KUKA KRL program: EPS_2_251806_MH03A_A_20260213065131.src

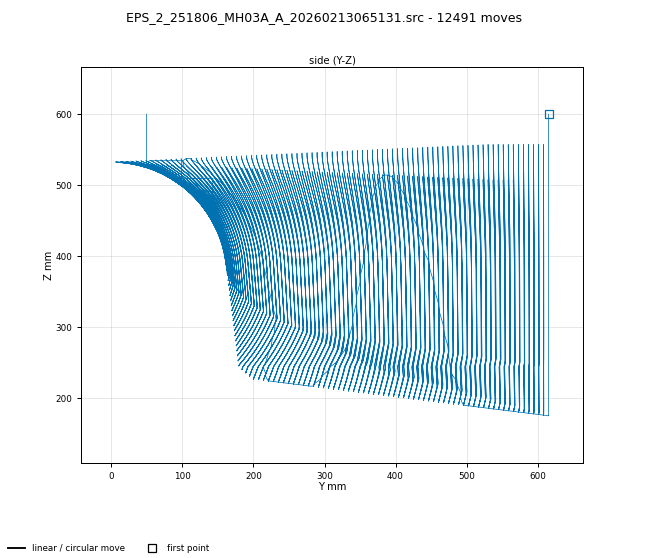
[picture p0: tool path of EPS_2_251806_MH03A_A_20260213065131.src, 12491 of 12493 moves have a stored position in this frame; points joined in program order, loops and branches not executed]
&ACCESS RVP
&REL 4
&COMMENT QRS 19112012
&PARAM EDITMASK = *
DEF PART()
EXT BAS (BAS_COMMAND :IN,REAL :IN )
INT I
BAS (#INITMOV,0 )

;KUKA QRS Post kuka4.cps  Date:22-06-2017 !

File_ID=3027

QRS_PRE_INIT()

;Init var - Until changes are made in qrs_pre_init
Outlet_Square_prg=0
Inlet_1_Square_prg=0
Inlet_2_Square_prg=0
Inlet_3_Square_prg=0
Inlet_4_Square_prg=0
Inlet_5_Square_prg=0

Outlet_1={X 0.000, Y 529.100, Z 408.000, B 0.000, E1 0.000 }
Inlet_1={X 0.000, Y 536.530, Z 382.000, B 0.000, E1 180.000 }
Outlet_1_type=299
Inlet_1_type=251
;QRS#1=Sidecore dimensions
;QRS#2=300-12" PVC SDR 35
;QRS#3=250-10" PVC SDR 35
;QRS#4=
;QRS#5=
;QRS#6=
;QRS#7=
;QRS#8=
;QRS#9=16M PSX
;QRS#10=14M PSX
;QRS#11=
;QRS#12=
;QRS#13=
;QRS#14=
;QRS#15=
;QRS#16=1220x127x838 2,75'
;QRS#17=EPS Height
;QRS#18=557,5
;QRS#19=*
;QRS#20= UPDATED VERSION 22-06-2017
;QRS#21=*
Outlet_Square=0150
Inlet_1_Square=0100
Inlet_2_Square=0
Inlet_3_Square=0
Inlet_4_Square=0
Inlet_5_Square=0
Mill_Square=1
Outlet_Square_Prg=206
Inlet_1_Square_prg=205

QRS_INIT()

$ADVANCE=5

; T1
PTP {E1 173.606,E2 173.606}
PTP {X 0,Y 615.5,A -85,B 0,C 180,E1 173.606,E2 173.606,E3 0,E4 0,E5 0,E6 0}
QRS_SPEED_INIT()
LIN {X 0,Y 615.5,Z 600,A -85,B 0,C 180,E1 173.606,E2 173.606,E3 0,E4 0,E5 0,E6 0} C_VEL
LIN {X 0,Y 615.5,Z 185.489,A -85,B 0,C 180,E1 173.606,E2 173.606} C_VEL
LIN {X 0,Y 615.5,Z 177.309,A -85,B 0,C 180,E1 173.606,E2 173.606} C_VEL
LIN {X 0,Y 615.485,Z 175.309,A -85,B 0,C 180,E1 173.419,E2 173.419} C_VEL
LIN {X 0,Y 615.484,Z 175.321,A -85,B 0,C 180,E1 170.801,E2 170.801} C_VEL
LIN {X 0,Y 615.479,Z 175.314,A -85,B 0,C 180,E1 168.139,E2 168.139} C_VEL
LIN {X 0,Y 615.481,Z 175.311,A -85,B 0,C 180,E1 165.451,E2 165.451} C_VEL
LIN {X 0,Y 615.493,Z 175.325,A -85,B 0,C 180,E1 162.73,E2 162.73} C_VEL
LIN {X 0,Y 615.49,Z 175.308,A -85,B 0,C 180,E1 159.967,E2 159.967} C_VEL
LIN {X 0,Y 615.483,Z 175.321,A -85,B 0,C 180,E1 157.155,E2 157.155} C_VEL
LIN {X 0,Y 615.475,Z 175.315,A -85,B 0,C 180,E1 154.433,E2 154.433} C_VEL
LIN {X 0,Y 615.483,Z 175.309,A -85,B 0,C 180,E1 152.085,E2 152.085} C_VEL
LIN {X 0,Y 615.492,Z 175.326,A -85,B 0,C 180,E1 149.08,E2 149.08} C_VEL
LIN {X 0,Y 615.474,Z 175.312,A -85,B 0,C 180,E1 146.467,E2 146.467} C_VEL
LIN {X 0,Y 615.492,Z 175.307,A -85,B 0,C 180,E1 144.165,E2 144.165} C_VEL
LIN {X 0,Y 615.485,Z 175.311,A -85,B 0,C 180,E1 141.931,E2 141.931} C_VEL
LIN {X 0,Y 615.486,Z 175.327,A -85,B 0,C 180,E1 139.393,E2 139.393} C_VEL
LIN {X 0,Y 615.469,Z 175.314,A -85,B 0,C 180,E1 136.753,E2 136.753} C_VEL
LIN {X 0,Y 615.488,Z 175.312,A -85,B 0,C 180,E1 133.997,E2 133.997} C_VEL
LIN {X 0,Y 615.49,Z 175.325,A -85,B 0,C 180,E1 131.473,E2 131.473} C_VEL
LIN {X 0,Y 615.465,Z 175.315,A -85,B 0,C 180,E1 128.906,E2 128.906} C_VEL
LIN {X 0,Y 615.484,Z 175.31,A -85,B 0,C 180,E1 126.425,E2 126.425} C_VEL
LIN {X 0,Y 615.481,Z 175.322,A -85,B 0,C 180,E1 123.533,E2 123.533} C_VEL
LIN {X 0,Y 615.466,Z 175.313,A -85,B 0,C 180,E1 120.921,E2 120.921} C_VEL
LIN {X 0,Y 615.493,Z 175.31,A -85,B 0,C 180,E1 118.451,E2 118.451} C_VEL
LIN {X 0,Y 615.468,Z 175.32,A -85,B 0,C 180,E1 115.565,E2 115.565} C_VEL
LIN {X 0,Y 615.491,Z 175.47,A -85,B 0,C 180,E1 113.895,E2 113.895} C_VEL
LIN {X 0,Y 615.494,Z 175.898,A -85,B 0,C 180,E1 113.782,E2 113.782} C_VEL
LIN {X 0,Y 615.488,Z 197.974,A -85,B 0,C 180,E1 111.081,E2 111.081} C_VEL
LIN {X 0,Y 615.498,Z 221.291,A -85,B 0,C 180,E1 108.281,E2 108.281} C_VEL
LIN {X 0,Y 615.478,Z 244.188,A -85,B 0,C 180,E1 105.587,E2 105.587} C_VEL
LIN {X 0,Y 615.48,Z 246.608,A -85,B 0,C 180,E1 105.523,E2 105.523} C_VEL
LIN {X 0,Y 615.498,Z 382.16,A -85,B 0,C 180,E1 103.905,E2 103.905} C_VEL
LIN {X 0,Y 615.497,Z 395.745,A -85,B 0,C 180,E1 103.621,E2 103.621} C_VEL
LIN {X 0,Y 615.497,Z 409.485,A -85,B 0,C 180,E1 103.201,E2 103.201} C_VEL
LIN {X 0,Y 615.492,Z 421.898,A -85,B 0,C 180,E1 102.698,E2 102.698} C_VEL
LIN {X 0,Y 615.486,Z 434.841,A -85,B 0,C 180,E1 102.028,E2 102.028} C_VEL
LIN {X 0,Y 615.499,Z 446.557,A -85,B 0,C 180,E1 101.276,E2 101.276} C_VEL
LIN {X 0,Y 615.498,Z 458.224,A -85,B 0,C 180,E1 100.361,E2 100.361} C_VEL
LIN {X 0,Y 615.497,Z 468.649,A -85,B 0,C 180,E1 99.364,E2 99.364} C_VEL
LIN {X 0,Y 615.496,Z 477.239,A -85,B 0,C 180,E1 98.371,E2 98.371} C_VEL
LIN {X 0,Y 615.495,Z 485.452,A -85,B 0,C 180,E1 97.216,E2 97.216} C_VEL
LIN {X 0,Y 615.496,Z 491.183,A -85,B 0,C 180,E1 96.228,E2 96.228} C_VEL
LIN {X 0,Y 615.494,Z 495.886,A -85,B 0,C 180,E1 95.241,E2 95.241} C_VEL
LIN {X 0,Y 615.496,Z 500.756,A -85,B 0,C 180,E1 93.929,E2 93.929} C_VEL
LIN {X 0,Y 615.496,Z 504.154,A -85,B 0,C 180,E1 92.618,E2 92.618} C_VEL
LIN {X 0,Y 615.493,Z 506.174,A -85,B 0,C 180,E1 91.309,E2 91.309} C_VEL
LIN {X 0,Y 615.494,Z 506.884,A -85,B 0,C 180,E1 90,E2 90} C_VEL
LIN {X 0,Y 615.49,Z 506.281,A -85,B 0,C 180,E1 88.692,E2 88.692} C_VEL
LIN {X 0,Y 615.493,Z 504.351,A -85,B 0,C 180,E1 87.382,E2 87.382} C_VEL
LIN {X 0,Y 615.496,Z 501.046,A -85,B 0,C 180,E1 86.072,E2 86.072} C_VEL
LIN {X 0,Y 615.496,Z 496.275,A -85,B 0,C 180,E1 84.759,E2 84.759} C_VEL
LIN {X 0,Y 615.494,Z 489.876,A -85,B 0,C 180,E1 83.444,E2 83.444} C_VEL
LIN {X 0,Y 615.496,Z 482.746,A -85,B 0,C 180,E1 82.29,E2 82.29} C_VEL
LIN {X 0,Y 615.497,Z 475.274,A -85,B 0,C 180,E1 81.298,E2 81.298} C_VEL
LIN {X 0,Y 615.496,Z 466.295,A -85,B 0,C 180,E1 80.304,E2 80.304} C_VEL
LIN {X 0,Y 615.498,Z 455.207,A -85,B 0,C 180,E1 79.291,E2 79.291} C_VEL
LIN {X 0,Y 615.498,Z 444.286,A -85,B 0,C 180,E1 78.474,E2 78.474} C_VEL
LIN {X 0,Y 615.486,Z 431.991,A -85,B 0,C 180,E1 77.721,E2 77.721} C_VEL
LIN {X 0,Y 615.494,Z 420.154,A -85,B 0,C 180,E1 77.135,E2 77.135} C_VEL
LIN {X 0,Y 615.495,Z 407.231,A -85,B 0,C 180,E1 76.631,E2 76.631} C_VEL
LIN {X 0,Y 615.498,Z 394.256,A -85,B 0,C 180,E1 76.253,E2 76.253} C_VEL
LIN {X 0,Y 615.497,Z 381.001,A -85,B 0,C 180,E1 75.988,E2 75.988} C_VEL
LIN {X 0,Y 615.479,Z 244.626,A -85,B 0,C 180,E1 74.35,E2 74.35} C_VEL
LIN {X 0,Y 615.486,Z 239.884,A -85,B 0,C 180,E1 73.831,E2 73.831} C_VEL
LIN {X 0,Y 615.488,Z 216.097,A -85,B 0,C 180,E1 71.009,E2 71.009} C_VEL
LIN {X 0,Y 615.477,Z 192.927,A -85,B 0,C 180,E1 68.216,E2 68.216} C_VEL
LIN {X 0,Y 615.496,Z 175.625,A -85,B 0,C 180,E1 66.075,E2 66.075} C_VEL
LIN {X 0,Y 615.494,Z 175.319,A -85,B 0,C 180,E1 65.729,E2 65.729} C_VEL
LIN {X 0,Y 615.455,Z 175.316,A -85,B 0,C 180,E1 62.822,E2 62.822} C_VEL
LIN {X 0,Y 615.487,Z 175.324,A -85,B 0,C 180,E1 60.206,E2 60.206} C_VEL
LIN {X 0,Y 615.493,Z 175.31,A -85,B 0,C 180,E1 57.544,E2 57.544} C_VEL
LIN {X 0,Y 615.466,Z 175.313,A -85,B 0,C 180,E1 55.184,E2 55.184} C_VEL
LIN {X 0,Y 615.463,Z 175.319,A -85,B 0,C 180,E1 52.757,E2 52.757} C_VEL
LIN {X 0,Y 615.488,Z 175.314,A -85,B 0,C 180,E1 49.911,E2 49.911} C_VEL
LIN {X 0,Y 615.494,Z 175.308,A -85,B 0,C 180,E1 47.649,E2 47.649} C_VEL
LIN {X 0,Y 615.466,Z 175.318,A -85,B 0,C 180,E1 44.931,E2 44.931} C_VEL
LIN {X 0,Y 615.488,Z 175.313,A -85,B 0,C 180,E1 42.081,E2 42.081} C_VEL
LIN {X 0,Y 615.488,Z 175.308,A -85,B 0,C 180,E1 39.75,E2 39.75} C_VEL
LIN {X 0,Y 615.475,Z 175.321,A -85,B 0,C 180,E1 36.937,E2 36.937} C_VEL
LIN {X 0,Y 615.489,Z 175.309,A -85,B 0,C 180,E1 34.022,E2 34.022} C_VEL
LIN {X 0,Y 615.477,Z 175.31,A -85,B 0,C 180,E1 31.686,E2 31.686} C_VEL
LIN {X 0,Y 615.469,Z 175.316,A -85,B 0,C 180,E1 29.407,E2 29.407} C_VEL
LIN {X 0,Y 615.488,Z 175.323,A -85,B 0,C 180,E1 27.047,E2 27.047} C_VEL
LIN {X 0,Y 615.489,Z 175.309,A -85,B 0,C 180,E1 24.272,E2 24.272} C_VEL
LIN {X 0,Y 615.476,Z 175.318,A -85,B 0,C 180,E1 21.432,E2 21.432} C_VEL
LIN {X 0,Y 615.481,Z 175.314,A -85,B 0,C 180,E1 18.606,E2 18.606} C_VEL
LIN {X 0,Y 615.476,Z 175.312,A -85,B 0,C 180,E1 15.906,E2 15.906} C_VEL
LIN {X 0,Y 615.495,Z 175.324,A -85,B 0,C 180,E1 13.201,E2 13.201} C_VEL
LIN {X 0,Y 615.486,Z 175.309,A -85,B 0,C 180,E1 10.527,E2 10.527} C_VEL
LIN {X 0,Y 615.479,Z 175.315,A -85,B 0,C 180,E1 7.876,E2 7.876} C_VEL
LIN {X 0,Y 615.484,Z 175.321,A -85,B 0,C 180,E1 5.241,E2 5.241} C_VEL
LIN {X 0,Y 615.487,Z 175.308,A -85,B 0,C 180,E1 2.618,E2 2.618} C_VEL
LIN {X 0,Y 615.479,Z 175.317,A -85,B 0,C 180,E1 0,E2 0} C_VEL
LIN {X 0,Y 615.479,Z 175.32,A -85,B 0,C 180,E1 -2.618,E2 -2.618} C_VEL
LIN {X 0,Y 615.485,Z 175.308,A -85,B 0,C 180,E1 -5.241,E2 -5.241} C_VEL
LIN {X 0,Y 615.485,Z 175.317,A -85,B 0,C 180,E1 -7.876,E2 -7.876} C_VEL
LIN {X 0,Y 615.472,Z 175.319,A -85,B 0,C 180,E1 -10.527,E2 -10.527} C_VEL
LIN {X 0,Y 615.492,Z 175.307,A -85,B 0,C 180,E1 -13.201,E2 -13.201} C_VEL
LIN {X 0,Y 615.491,Z 175.323,A -85,B 0,C 180,E1 -15.905,E2 -15.905} C_VEL
LIN {X 0,Y 615.465,Z 175.315,A -85,B 0,C 180,E1 -18.647,E2 -18.647} C_VEL
LIN {X 0,Y 615.486,Z 175.314,A -85,B 0,C 180,E1 -21.432,E2 -21.432} C_VEL
LIN {X 0,Y 615.466,Z 175.318,A -85,B 0,C 180,E1 -24.273,E2 -24.273} C_VEL
LIN {X 0,Y 615.497,Z 175.308,A -85,B 0,C 180,E1 -27.049,E2 -27.049} C_VEL
LIN {X 0,Y 615.485,Z 175.324,A -85,B 0,C 180,E1 -29.796,E2 -29.796} C_VEL
LIN {X 0,Y 615.46,Z 175.314,A -85,B 0,C 180,E1 -32.459,E2 -32.459} C_VEL
LIN {X 0,Y 615.487,Z 175.309,A -85,B 0,C 180,E1 -34.815,E2 -34.815} C_VEL
LIN {X 0,Y 615.492,Z 175.318,A -85,B 0,C 180,E1 -37.242,E2 -37.242} C_VEL
LIN {X 0,Y 615.468,Z 175.321,A -85,B 0,C 180,E1 -39.752,E2 -39.752} C_VEL
LIN {X 0,Y 615.46,Z 175.314,A -85,B 0,C 180,E1 -42.355,E2 -42.355} C_VEL
LIN {X 0,Y 615.489,Z 175.32,A -85,B 0,C 180,E1 -45.068,E2 -45.068} C_VEL
LIN {X 0,Y 615.456,Z 175.322,A -85,B 0,C 180,E1 -47.645,E2 -47.645} C_VEL
LIN {X 0,Y 615.459,Z 175.314,A -85,B 0,C 180,E1 -50.249,E2 -50.249} C_VEL
LIN {X 0,Y 615.487,Z 175.327,A -85,B 0,C 180,E1 -53.063,E2 -53.063} C_VEL
LIN {X 0,Y 615.47,Z 175.323,A -85,B 0,C 180,E1 -55.302,E2 -55.302} C_VEL
LIN {X 0,Y 615.446,Z 175.319,A -85,B 0,C 180,E1 -57.675,E2 -57.675} C_VEL
LIN {X 0,Y 615.462,Z 175.315,A -85,B 0,C 180,E1 -60.209,E2 -60.209} C_VEL
LIN {X 0,Y 615.486,Z 175.324,A -85,B 0,C 180,E1 -62.955,E2 -62.955} C_VEL
LIN {X 0,Y 615.497,Z 175.476,A -85,B 0,C 180,E1 -64.901,E2 -64.901} C_VEL
LIN {X 0,Y 615.497,Z 176.063,A -85,B 0,C 180,E1 -65.009,E2 -65.009} C_VEL
LIN {X 0,Y 615.436,Z 201.512,A -85,B 0,C 180,E1 -67.537,E2 -67.537} C_VEL
LIN {X 0,Y 615.488,Z 230.015,A -85,B 0,C 180,E1 -70.316,E2 -70.316} C_VEL
LIN {X 0,Y 615.494,Z 245.089,A -85,B 0,C 180,E1 -71.741,E2 -71.741} C_VEL
LIN {X 0,Y 615.498,Z 411.933,A -85,B 0,C 180,E1 -73.765,E2 -73.765} C_VEL
LIN {X 0,Y 615.497,Z 427.732,A -85,B 0,C 180,E1 -74.096,E2 -74.096} C_VEL
LIN {X 0,Y 615.481,Z 443.064,A -85,B 0,C 180,E1 -74.562,E2 -74.562} C_VEL
LIN {X 0,Y 615.494,Z 456.765,A -85,B 0,C 180,E1 -75.113,E2 -75.113} C_VEL
LIN {X 0,Y 615.495,Z 471.049,A -85,B 0,C 180,E1 -75.834,E2 -75.834} C_VEL
LIN {X 0,Y 615.497,Z 483.905,A -85,B 0,C 180,E1 -76.631,E2 -76.631} C_VEL
LIN {X 0,Y 615.495,Z 496.26,A -85,B 0,C 180,E1 -77.554,E2 -77.554} C_VEL
LIN {X 0,Y 615.495,Z 506.611,A -85,B 0,C 180,E1 -78.474,E2 -78.474} C_VEL
LIN {X 0,Y 615.495,Z 516.188,A -85,B 0,C 180,E1 -79.474,E2 -79.474} C_VEL
LIN {X 0,Y 615.493,Z 525.58,A -85,B 0,C 180,E1 -80.636,E2 -80.636} C_VEL
LIN {X 0,Y 615.494,Z 533.383,A -85,B 0,C 180,E1 -81.794,E2 -81.794} C_VEL
LIN {X 0,Y 615.496,Z 540.607,A -85,B 0,C 180,E1 -83.102,E2 -83.102} C_VEL
LIN {X 0,Y 615.499,Z 546.438,A -85,B 0,C 180,E1 -84.431,E2 -84.431} C_VEL
LIN {X 0,Y 615.491,Z 549.861,A -85,B 0,C 180,E1 -85.416,E2 -85.416} C_VEL
LIN {X 0,Y 615.492,Z 553.319,A -85,B 0,C 180,E1 -86.727,E2 -86.727} C_VEL
LIN {X 0,Y 615.499,Z 555.593,A -85,B 0,C 180,E1 -88.037,E2 -88.037} C_VEL
LIN {X 0,Y 615.494,Z 556.74,A -85,B 0,C 180,E1 -89.346,E2 -89.346} C_VEL
LIN {X 0,Y 615.494,Z 556.74,A -85,B 0,C 180,E1 -90.654,E2 -90.654} C_VEL
LIN {X 0,Y 615.499,Z 555.592,A -85,B 0,C 180,E1 -91.963,E2 -91.963} C_VEL
LIN {X 0,Y 615.492,Z 553.318,A -85,B 0,C 180,E1 -93.273,E2 -93.273} C_VEL
LIN {X 0,Y 615.491,Z 549.86,A -85,B 0,C 180,E1 -94.585,E2 -94.585} C_VEL
LIN {X 0,Y 615.499,Z 545.141,A -85,B 0,C 180,E1 -95.899,E2 -95.899} C_VEL
LIN {X 0,Y 615.494,Z 539.028,A -85,B 0,C 180,E1 -97.216,E2 -97.216} C_VEL
LIN {X 0,Y 615.494,Z 531.331,A -85,B 0,C 180,E1 -98.537,E2 -98.537} C_VEL
LIN {X 0,Y 615.495,Z 523.113,A -85,B 0,C 180,E1 -99.696,E2 -99.696} C_VEL
LIN {X 0,Y 615.497,Z 512.891,A -85,B 0,C 180,E1 -100.893,E2 -100.893} C_VEL
LIN {X 0,Y 615.495,Z 503.066,A -85,B 0,C 180,E1 -101.861,E2 -101.861} C_VEL
LIN {X 0,Y 615.497,Z 490.946,A -85,B 0,C 180,E1 -102.865,E2 -102.865} C_VEL
LIN {X 0,Y 615.498,Z 478.796,A -85,B 0,C 180,E1 -103.706,E2 -103.706} C_VEL
LIN {X 0,Y 615.488,Z 465.377,A -85,B 0,C 180,E1 -104.472,E2 -104.472} C_VEL
LIN {X 0,Y 615.494,Z 450.847,A -85,B 0,C 180,E1 -105.141,E2 -105.141} C_VEL
LIN {X 0,Y 615.495,Z 436.614,A -85,B 0,C 180,E1 -105.65,E2 -105.65} C_VEL
LIN {X 0,Y 615.5,Z 422.078,A -85,B 0,C 180,E1 -106.037,E2 -106.037} C_VEL
LIN {X 0,Y 615.498,Z 407.298,A -85,B 0,C 180,E1 -106.301,E2 -106.301} C_VEL
LIN {X 0,Y 615.492,Z 245.082,A -85,B 0,C 180,E1 -108.259,E2 -108.259} C_VEL
LIN {X 0,Y 615.451,Z 221.108,A -85,B 0,C 180,E1 -110.548,E2 -110.548} C_VEL
LIN {X 0,Y 615.453,Z 195.818,A -85,B 0,C 180,E1 -113.023,E2 -113.023} C_VEL
LIN {X 0,Y 615.498,Z 175.662,A -85,B 0,C 180,E1 -115.045,E2 -115.045} C_VEL
LIN {X 0,Y 615.498,Z 175.313,A -85,B 0,C 180,E1 -115.571,E2 -115.571} C_VEL
LIN {X 0,Y 615.458,Z 175.315,A -85,B 0,C 180,E1 -117.916,E2 -117.916} C_VEL
LIN {X 0,Y 615.446,Z 175.317,A -85,B 0,C 180,E1 -120.162,E2 -120.162} C_VEL
LIN {X 0,Y 615.449,Z 175.32,A -85,B 0,C 180,E1 -122.46,E2 -122.46} C_VEL
LIN {X 0,Y 615.48,Z 175.324,A -85,B 0,C 180,E1 -124.815,E2 -124.815} C_VEL
LIN {X 0,Y 615.493,Z 175.316,A -85,B 0,C 180,E1 -127.241,E2 -127.241} C_VEL
LIN {X 0,Y 615.458,Z 175.315,A -85,B 0,C 180,E1 -129.752,E2 -129.752} C_VEL
LIN {X 0,Y 615.457,Z 175.321,A -85,B 0,C 180,E1 -132.355,E2 -132.355} C_VEL
LIN {X 0,Y 615.488,Z 175.316,A -85,B 0,C 180,E1 -135.068,E2 -135.068} C_VEL
LIN {X 0,Y 615.459,Z 175.314,A -85,B 0,C 180,E1 -137.645,E2 -137.645} C_VEL
LIN {X 0,Y 615.466,Z 175.321,A -85,B 0,C 180,E1 -140.248,E2 -140.248} C_VEL
LIN {X 0,Y 615.487,Z 175.312,A -85,B 0,C 180,E1 -143.063,E2 -143.063} C_VEL
LIN {X 0,Y 615.477,Z 175.311,A -85,B 0,C 180,E1 -145.3,E2 -145.3} C_VEL
LIN {X 0,Y 615.457,Z 175.316,A -85,B 0,C 180,E1 -147.673,E2 -147.673} C_VEL
LIN {X 0,Y 615.483,Z 175.324,A -85,B 0,C 180,E1 -150.205,E2 -150.205} C_VEL
LIN {X 0,Y 615.497,Z 175.308,A -85,B 0,C 180,E1 -152.952,E2 -152.952} C_VEL
LIN {X 0,Y 615.464,Z 175.318,A -85,B 0,C 180,E1 -155.727,E2 -155.727} C_VEL
LIN {X 0,Y 615.487,Z 175.315,A -85,B 0,C 180,E1 -158.568,E2 -158.568} C_VEL
LIN {X 0,Y 615.462,Z 175.316,A -85,B 0,C 180,E1 -161.401,E2 -161.401} C_VEL
LIN {X 0,Y 615.488,Z 175.325,A -85,B 0,C 180,E1 -164.095,E2 -164.095} C_VEL
LIN {X 0,Y 615.492,Z 175.307,A -85,B 0,C 180,E1 -166.799,E2 -166.799} C_VEL
LIN {X 0,Y 615.47,Z 175.319,A -85,B 0,C 180,E1 -169.473,E2 -169.473} C_VEL
LIN {X 0,Y 615.486,Z 175.318,A -85,B 0,C 180,E1 -172.124,E2 -172.124} C_VEL
LIN {X 0,Y 615.485,Z 175.308,A -85,B 0,C 180,E1 -174.759,E2 -174.759} C_VEL
LIN {X 0,Y 615.473,Z 175.321,A -85,B 0,C 180,E1 -177.382,E2 -177.382} C_VEL
LIN {X 0,Y 615.484,Z 175.317,A -85,B 0,C 180,E1 -180,E2 -180} C_VEL
LIN {X 0,Y 615.486,Z 175.308,A -85,B 0,C 180,E1 -182.618,E2 -182.618} C_VEL
LIN {X 0,Y 615.48,Z 175.32,A -85,B 0,C 180,E1 -185.241,E2 -185.241} C_VEL
LIN {X 0,Y 615.485,Z 175.309,A -85,B 0,C 180,E1 -186.581,E2 -186.581} C_VEL
LIN {X 0,Y 614.808,Z 175.467,A -85,B 0,C 180,E1 -187.127,E2 -187.127} C_VEL
LIN {X 0,Y 611.973,Z 175.876,A -85,B 0,C 180,E1 -188.013,E2 -188.013} C_VEL
LIN {X 0,Y 609.582,Z 176.191,A -85,B 0,C 180,E1 -188.725,E2 -188.725} C_VEL
LIN {X 0,Y 608.546,Z 176.31,A -85,B 0,C 180,E1 -189.275,E2 -189.275} C_VEL
LIN {X 0,Y 608.456,Z 176.318,A -85,B 0,C 180,E1 -189.461,E2 -189.461} C_VEL
LIN {X 0,Y 608.456,Z 176.313,A -85,B 0,C 180,E1 -192,E2 -192} C_VEL
LIN {X 0,Y 608.471,Z 176.312,A -85,B 0,C 180,E1 -194.721,E2 -194.721} C_VEL
LIN {X 0,Y 608.455,Z 176.318,A -85,B 0,C 180,E1 -197.477,E2 -197.477} C_VEL
LIN {X 0,Y 608.461,Z 176.312,A -85,B 0,C 180,E1 -200.274,E2 -200.274} C_VEL
LIN {X 0,Y 608.456,Z 176.314,A -85,B 0,C 180,E1 -202.477,E2 -202.477} C_VEL
LIN {X 0,Y 608.456,Z 176.315,A -85,B 0,C 180,E1 -204.571,E2 -204.571} C_VEL
LIN {X 0,Y 608.479,Z 176.315,A -85,B 0,C 180,E1 -207.208,E2 -207.208} C_VEL
LIN {X 0,Y 608.467,Z 176.311,A -85,B 0,C 180,E1 -209.972,E2 -209.972} C_VEL
LIN {X 0,Y 608.45,Z 176.323,A -85,B 0,C 180,E1 -212.88,E2 -212.88} C_VEL
LIN {X 0,Y 608.443,Z 176.316,A -85,B 0,C 180,E1 -215.278,E2 -215.278} C_VEL
LIN {X 0,Y 608.466,Z 176.314,A -85,B 0,C 180,E1 -218.241,E2 -218.241} C_VEL
LIN {X 0,Y 608.45,Z 176.314,A -85,B 0,C 180,E1 -221.341,E2 -221.341} C_VEL
LIN {X 0,Y 608.453,Z 176.318,A -85,B 0,C 180,E1 -224.264,E2 -224.264} C_VEL
LIN {X 0,Y 608.439,Z 176.316,A -85,B 0,C 180,E1 -227.039,E2 -227.039} C_VEL
LIN {X 0,Y 608.452,Z 176.313,A -85,B 0,C 180,E1 -229.697,E2 -229.697} C_VEL
LIN {X 0,Y 608.465,Z 176.32,A -85,B 0,C 180,E1 -232.254,E2 -232.254} C_VEL
LIN {X 0,Y 608.437,Z 176.315,A -85,B 0,C 180,E1 -235.096,E2 -235.096} C_VEL
LIN {X 0,Y 608.471,Z 176.315,A -85,B 0,C 180,E1 -237.906,E2 -237.906} C_VEL
LIN {X 0,Y 608.481,Z 176.319,A -85,B 0,C 180,E1 -240.221,E2 -240.221} C_VEL
LIN {X 0,Y 608.438,Z 176.316,A -85,B 0,C 180,E1 -242.801,E2 -242.801} C_VEL
LIN {X 0,Y 608.449,Z 176.316,A -85,B 0,C 180,E1 -245.429,E2 -245.429} C_VEL
LIN {X 0,Y 608.511,Z 176.616,A -85,B 0,C 180,E1 -246.014,E2 -246.014} C_VEL
LIN {X 0,Y 608.609,Z 190.74,A -85,B 0,C 180,E1 -247.779,E2 -247.779} C_VEL
LIN {X 0,Y 608.566,Z 212.456,A -85,B 0,C 180,E1 -250.433,E2 -250.433} C_VEL
LIN {X 0,Y 608.529,Z 235.621,A -85,B 0,C 180,E1 -253.218,E2 -253.218} C_VEL
LIN {X 0,Y 608.522,Z 244.516,A -85,B 0,C 180,E1 -254.252,E2 -254.252} C_VEL
LIN {X 0,Y 608.658,Z 255.594,A -85,B 0,C 180,E1 -254.406,E2 -254.406} C_VEL
LIN {X 0,Y 608.609,Z 382.975,A -85,B 0,C 180,E1 -255.949,E2 -255.949} C_VEL
LIN {X 0,Y 608.613,Z 397.296,A -85,B 0,C 180,E1 -256.264,E2 -256.264} C_VEL
LIN {X 0,Y 608.586,Z 410.642,A -85,B 0,C 180,E1 -256.689,E2 -256.689} C_VEL
LIN {X 0,Y 608.542,Z 423.702,A -85,B 0,C 180,E1 -257.24,E2 -257.24} C_VEL
LIN {X 0,Y 608.529,Z 436.34,A -85,B 0,C 180,E1 -257.917,E2 -257.917} C_VEL
LIN {X 0,Y 608.5,Z 447.85,A -85,B 0,C 180,E1 -258.677,E2 -258.677} C_VEL
LIN {X 0,Y 608.495,Z 458.411,A -85,B 0,C 180,E1 -259.519,E2 -259.519} C_VEL
LIN {X 0,Y 608.48,Z 468.897,A -85,B 0,C 180,E1 -260.527,E2 -260.527} C_VEL
LIN {X 0,Y 608.463,Z 477.55,A -85,B 0,C 180,E1 -261.531,E2 -261.531} C_VEL
LIN {X 0,Y 608.46,Z 485.838,A -85,B 0,C 180,E1 -262.7,E2 -262.7} C_VEL
LIN {X 0,Y 608.443,Z 492.324,A -85,B 0,C 180,E1 -263.831,E2 -263.831} C_VEL
LIN {X 0,Y 608.435,Z 497.787,A -85,B 0,C 180,E1 -265.03,E2 -265.03} C_VEL
LIN {X 0,Y 608.434,Z 501.297,A -85,B 0,C 180,E1 -266.026,E2 -266.026} C_VEL
LIN {X 0,Y 608.424,Z 504.733,A -85,B 0,C 180,E1 -267.352,E2 -267.352} C_VEL
LIN {X 0,Y 608.446,Z 506.777,A -85,B 0,C 180,E1 -268.676,E2 -268.676} C_VEL
LIN {X 0,Y 608.434,Z 507.495,A -85,B 0,C 180,E1 -270,E2 -270} C_VEL
LIN {X 0,Y 608.443,Z 506.883,A -85,B 0,C 180,E1 -271.323,E2 -271.323} C_VEL
LIN {X 0,Y 608.421,Z 504.929,A -85,B 0,C 180,E1 -272.648,E2 -272.648} C_VEL
LIN {X 0,Y 608.434,Z 501.586,A -85,B 0,C 180,E1 -273.974,E2 -273.974} C_VEL
LIN {X 0,Y 608.44,Z 496.761,A -85,B 0,C 180,E1 -275.302,E2 -275.302} C_VEL
LIN {X 0,Y 608.442,Z 490.474,A -85,B 0,C 180,E1 -276.6,E2 -276.6} C_VEL
LIN {X 0,Y 608.453,Z 483.102,A -85,B 0,C 180,E1 -277.8,E2 -277.8} C_VEL
LIN {X 0,Y 608.476,Z 475.566,A -85,B 0,C 180,E1 -278.803,E2 -278.803} C_VEL
LIN {X 0,Y 608.488,Z 466.522,A -85,B 0,C 180,E1 -279.808,E2 -279.808} C_VEL
LIN {X 0,Y 608.506,Z 455.723,A -85,B 0,C 180,E1 -280.804,E2 -280.804} C_VEL
LIN {X 0,Y 608.523,Z 444.389,A -85,B 0,C 180,E1 -281.66,E2 -281.66} C_VEL
LIN {X 0,Y 608.539,Z 432.048,A -85,B 0,C 180,E1 -282.421,E2 -282.421} C_VEL
LIN {X 0,Y 608.559,Z 420.181,A -85,B 0,C 180,E1 -283.014,E2 -283.014} C_VEL
LIN {X 0,Y 608.581,Z 407.232,A -85,B 0,C 180,E1 -283.523,E2 -283.523} C_VEL
LIN {X 0,Y 608.593,Z 392.998,A -85,B 0,C 180,E1 -283.935,E2 -283.935} C_VEL
LIN {X 0,Y 608.609,Z 378.849,A -85,B 0,C 180,E1 -284.204,E2 -284.204} C_VEL
LIN {X 0,Y 608.567,Z 244.888,A -85,B 0,C 180,E1 -285.822,E2 -285.822} C_VEL
LIN {X 0,Y 608.518,Z 243.627,A -85,B 0,C 180,E1 -285.92,E2 -285.92} C_VEL
LIN {X 0,Y 608.558,Z 222.058,A -85,B 0,C 180,E1 -288.497,E2 -288.497} C_VEL
LIN {X 0,Y 608.594,Z 197.268,A -85,B 0,C 180,E1 -291.508,E2 -291.508} C_VEL
LIN {X 0,Y 608.632,Z 178.436,A -85,B 0,C 180,E1 -293.837,E2 -293.837} C_VEL
LIN {X 0,Y 608.485,Z 176.516,A -85,B 0,C 180,E1 -294.108,E2 -294.108} C_VEL
LIN {X 0,Y 608.437,Z 176.315,A -85,B 0,C 180,E1 -296.774,E2 -296.774} C_VEL
LIN {X 0,Y 608.428,Z 176.316,A -85,B 0,C 180,E1 -299.021,E2 -299.021} C_VEL
LIN {X 0,Y 608.438,Z 176.317,A -85,B 0,C 180,E1 -301.317,E2 -301.317} C_VEL
LIN {X 0,Y 608.47,Z 176.319,A -85,B 0,C 180,E1 -303.734,E2 -303.734} C_VEL
LIN {X 0,Y 608.476,Z 176.314,A -85,B 0,C 180,E1 -306.089,E2 -306.089} C_VEL
LIN {X 0,Y 608.457,Z 176.312,A -85,B 0,C 180,E1 -308.588,E2 -308.588} C_VEL
LIN {X 0,Y 608.451,Z 176.318,A -85,B 0,C 180,E1 -311.341,E2 -311.341} C_VEL
LIN {X 0,Y 608.459,Z 176.313,A -85,B 0,C 180,E1 -314.264,E2 -314.264} C_VEL
LIN {X 0,Y 608.435,Z 176.318,A -85,B 0,C 180,E1 -317.038,E2 -317.038} C_VEL
LIN {X 0,Y 608.453,Z 176.318,A -85,B 0,C 180,E1 -319.697,E2 -319.697} C_VEL
LIN {X 0,Y 608.463,Z 176.311,A -85,B 0,C 180,E1 -322.253,E2 -322.253} C_VEL
LIN {X 0,Y 608.48,Z 176.316,A -85,B 0,C 180,E1 -325.089,E2 -325.089} C_VEL
LIN {X 0,Y 608.461,Z 176.313,A -85,B 0,C 180,E1 -327.905,E2 -327.905} C_VEL
LIN {X 0,Y 608.467,Z 176.311,A -85,B 0,C 180,E1 -330.22,E2 -330.22} C_VEL
LIN {X 0,Y 608.474,Z 176.315,A -85,B 0,C 180,E1 -332.791,E2 -332.791} C_VEL
LIN {X 0,Y 608.48,Z 176.309,A -85,B 0,C 180,E1 -335.845,E2 -335.845} C_VEL
LIN {X 0,Y 608.465,Z 176.312,A -85,B 0,C 180,E1 -338.308,E2 -338.308} C_VEL
LIN {X 0,Y 608.45,Z 176.319,A -85,B 0,C 180,E1 -341.13,E2 -341.13} C_VEL
LIN {X 0,Y 608.454,Z 176.312,A -85,B 0,C 180,E1 -343.906,E2 -343.906} C_VEL
LIN {X 0,Y 608.467,Z 176.32,A -85,B 0,C 180,E1 -346.644,E2 -346.644} C_VEL
LIN {X 0,Y 608.461,Z 176.313,A -85,B 0,C 180,E1 -349.35,E2 -349.35} C_VEL
LIN {X 0,Y 608.471,Z 176.312,A -85,B 0,C 180,E1 -352.033,E2 -352.033} C_VEL
LIN {X 0,Y 608.463,Z 176.319,A -85,B 0,C 180,E1 -354.698,E2 -354.698} C_VEL
LIN {X 0,Y 608.477,Z 176.31,A -85,B 0,C 180,E1 -357.352,E2 -357.352} C_VEL
LIN {X 0,Y 608.47,Z 176.314,A -85,B 0,C 180,E1 -360,E2 -360} C_VEL
LIN {X 0,Y 608.47,Z 176.316,A -85,B 0,C 180,E1 -362.648,E2 -362.648} C_VEL
LIN {X 0,Y 608.464,Z 176.311,A -85,B 0,C 180,E1 -365.302,E2 -365.302} C_VEL
LIN {X 0,Y 608.474,Z 176.316,A -85,B 0,C 180,E1 -367.967,E2 -367.967} C_VEL
LIN {X 0,Y 608.451,Z 176.315,A -85,B 0,C 180,E1 -370.65,E2 -370.65} C_VEL
LIN {X 0,Y 608.469,Z 176.311,A -85,B 0,C 180,E1 -373.356,E2 -373.356} C_VEL
LIN {X 0,Y 608.457,Z 176.321,A -85,B 0,C 180,E1 -376.094,E2 -376.094} C_VEL
LIN {X 0,Y 608.445,Z 176.313,A -85,B 0,C 180,E1 -378.87,E2 -378.87} C_VEL
LIN {X 0,Y 608.464,Z 176.318,A -85,B 0,C 180,E1 -381.692,E2 -381.692} C_VEL
LIN {X 0,Y 608.444,Z 176.314,A -85,B 0,C 180,E1 -384.571,E2 -384.571} C_VEL
LIN {X 0,Y 608.484,Z 176.311,A -85,B 0,C 180,E1 -387.21,E2 -387.21} C_VEL
LIN {X 0,Y 608.442,Z 176.319,A -85,B 0,C 180,E1 -389.969,E2 -389.969} C_VEL
LIN {X 0,Y 608.439,Z 176.314,A -85,B 0,C 180,E1 -392.521,E2 -392.521} C_VEL
LIN {X 0,Y 608.478,Z 176.311,A -85,B 0,C 180,E1 -394.911,E2 -394.911} C_VEL
LIN {X 0,Y 608.454,Z 176.318,A -85,B 0,C 180,E1 -397.747,E2 -397.747} C_VEL
LIN {X 0,Y 608.429,Z 176.316,A -85,B 0,C 180,E1 -400.328,E2 -400.328} C_VEL
LIN {X 0,Y 608.454,Z 176.316,A -85,B 0,C 180,E1 -402.96,E2 -402.96} C_VEL
LIN {X 0,Y 608.43,Z 176.318,A -85,B 0,C 180,E1 -405.739,E2 -405.739} C_VEL
LIN {X 0,Y 608.43,Z 176.316,A -85,B 0,C 180,E1 -407.937,E2 -407.937} C_VEL
LIN {X 0,Y 608.444,Z 176.316,A -85,B 0,C 180,E1 -410.705,E2 -410.705} C_VEL
LIN {X 0,Y 608.455,Z 176.323,A -85,B 0,C 180,E1 -413.086,E2 -413.086} C_VEL
LIN {X 0,Y 608.449,Z 176.316,A -85,B 0,C 180,E1 -415.53,E2 -415.53} C_VEL
LIN {X 0,Y 608.439,Z 176.314,A -85,B 0,C 180,E1 -417.905,E2 -417.905} C_VEL
LIN {X 0,Y 608.461,Z 176.321,A -85,B 0,C 180,E1 -420.98,E2 -420.98} C_VEL
LIN {X 0,Y 608.429,Z 176.322,A -85,B 0,C 180,E1 -423.225,E2 -423.225} C_VEL
LIN {X 0,Y 608.504,Z 176.484,A -85,B 0,C 180,E1 -424.725,E2 -424.725} C_VEL
LIN {X 0,Y 608.739,Z 179.627,A -85,B 0,C 180,E1 -425.078,E2 -425.078} C_VEL
LIN {X 0,Y 608.636,Z 206.621,A -85,B 0,C 180,E1 -427.78,E2 -427.78} C_VEL
LIN {X 0,Y 608.589,Z 235.414,A -85,B 0,C 180,E1 -430.61,E2 -430.61} C_VEL
LIN {X 0,Y 608.606,Z 245.087,A -85,B 0,C 180,E1 -431.527,E2 -431.527} C_VEL
LIN {X 0,Y 608.747,Z 290.93,A -85,B 0,C 180,E1 -432.099,E2 -432.099} C_VEL
LIN {X 0,Y 608.692,Z 411.932,A -85,B 0,C 180,E1 -433.578,E2 -433.578} C_VEL
LIN {X 0,Y 608.657,Z 427.73,A -85,B 0,C 180,E1 -433.912,E2 -433.912} C_VEL
LIN {X 0,Y 608.629,Z 443.062,A -85,B 0,C 180,E1 -434.384,E2 -434.384} C_VEL
LIN {X 0,Y 608.601,Z 456.768,A -85,B 0,C 180,E1 -434.941,E2 -434.941} C_VEL
LIN {X 0,Y 608.578,Z 470.245,A -85,B 0,C 180,E1 -435.625,E2 -435.625} C_VEL
LIN {X 0,Y 608.554,Z 482.671,A -85,B 0,C 180,E1 -436.391,E2 -436.391} C_VEL
LIN {X 0,Y 608.528,Z 495.289,A -85,B 0,C 180,E1 -437.325,E2 -437.325} C_VEL
LIN {X 0,Y 608.496,Z 506.752,A -85,B 0,C 180,E1 -438.339,E2 -438.339} C_VEL
LIN {X 0,Y 608.477,Z 516.392,A -85,B 0,C 180,E1 -439.351,E2 -439.351} C_VEL
LIN {X 0,Y 608.476,Z 525.857,A -85,B 0,C 180,E1 -440.527,E2 -440.527} C_VEL
LIN {X 0,Y 608.456,Z 533.732,A -85,B 0,C 180,E1 -441.699,E2 -441.699} C_VEL
LIN {X 0,Y 608.441,Z 541.089,A -85,B 0,C 180,E1 -443.034,E2 -443.034} C_VEL
LIN {X 0,Y 608.45,Z 546.925,A -85,B 0,C 180,E1 -444.366,E2 -444.366} C_VEL
LIN {X 0,Y 608.427,Z 550.384,A -85,B 0,C 180,E1 -445.362,E2 -445.362} C_VEL
LIN {X 0,Y 608.421,Z 553.886,A -85,B 0,C 180,E1 -446.689,E2 -446.689} C_VEL
LIN {X 0,Y 608.444,Z 556.192,A -85,B 0,C 180,E1 -448.014,E2 -448.014} C_VEL
LIN {X 0,Y 608.436,Z 557.351,A -85,B 0,C 180,E1 -449.338,E2 -449.338} C_VEL
LIN {X 0,Y 608.436,Z 557.35,A -85,B 0,C 180,E1 -450.662,E2 -450.662} C_VEL
LIN {X 0,Y 608.444,Z 556.191,A -85,B 0,C 180,E1 -451.986,E2 -451.986} C_VEL
LIN {X 0,Y 608.421,Z 553.885,A -85,B 0,C 180,E1 -453.311,E2 -453.311} C_VEL
LIN {X 0,Y 608.427,Z 550.382,A -85,B 0,C 180,E1 -454.638,E2 -454.638} C_VEL
LIN {X 0,Y 608.437,Z 545.607,A -85,B 0,C 180,E1 -455.967,E2 -455.967} C_VEL
LIN {X 0,Y 608.457,Z 539.425,A -85,B 0,C 180,E1 -457.3,E2 -457.3} C_VEL
LIN {X 0,Y 608.468,Z 531.653,A -85,B 0,C 180,E1 -458.636,E2 -458.636} C_VEL
LIN {X 0,Y 608.471,Z 523.369,A -85,B 0,C 180,E1 -459.809,E2 -459.809} C_VEL
LIN {X 0,Y 608.493,Z 512.647,A -85,B 0,C 180,E1 -461.063,E2 -461.063} C_VEL
LIN {X 0,Y 608.522,Z 501.273,A -85,B 0,C 180,E1 -462.168,E2 -462.168} C_VEL
LIN {X 0,Y 608.547,Z 489.853,A -85,B 0,C 180,E1 -463.1,E2 -463.1} C_VEL
LIN {X 0,Y 608.563,Z 477.446,A -85,B 0,C 180,E1 -463.95,E2 -463.95} C_VEL
LIN {X 0,Y 608.575,Z 463.858,A -85,B 0,C 180,E1 -464.718,E2 -464.718} C_VEL
LIN {X 0,Y 608.609,Z 449.79,A -85,B 0,C 180,E1 -465.359,E2 -465.359} C_VEL
LIN {X 0,Y 608.662,Z 434.565,A -85,B 0,C 180,E1 -465.895,E2 -465.895} C_VEL
LIN {X 0,Y 608.679,Z 419.085,A -85,B 0,C 180,E1 -466.288,E2 -466.288} C_VEL
LIN {X 0,Y 608.702,Z 404.275,A -85,B 0,C 180,E1 -466.531,E2 -466.531} C_VEL
LIN {X 0,Y 608.646,Z 245.405,A -85,B 0,C 180,E1 -468.461,E2 -468.461} C_VEL
LIN {X 0,Y 608.576,Z 240.808,A -85,B 0,C 180,E1 -468.866,E2 -468.866} C_VEL
LIN {X 0,Y 608.651,Z 212.014,A -85,B 0,C 180,E1 -471.685,E2 -471.685} C_VEL
LIN {X 0,Y 608.719,Z 183.221,A -85,B 0,C 180,E1 -474.56,E2 -474.56} C_VEL
LIN {X 0,Y 608.552,Z 176.75,A -85,B 0,C 180,E1 -475.228,E2 -475.228} C_VEL
LIN {X 0,Y 608.492,Z 176.334,A -85,B 0,C 180,E1 -475.372,E2 -475.372} C_VEL
LIN {X 0,Y 608.44,Z 176.319,A -85,B 0,C 180,E1 -477.518,E2 -477.518} C_VEL
LIN {X 0,Y 608.426,Z 176.313,A -85,B 0,C 180,E1 -479.965,E2 -479.965} C_VEL
LIN {X 0,Y 608.431,Z 176.318,A -85,B 0,C 180,E1 -482.518,E2 -482.518} C_VEL
LIN {X 0,Y 608.435,Z 176.32,A -85,B 0,C 180,E1 -485.278,E2 -485.278} C_VEL
LIN {X 0,Y 608.449,Z 176.313,A -85,B 0,C 180,E1 -487.747,E2 -487.747} C_VEL
LIN {X 0,Y 608.43,Z 176.317,A -85,B 0,C 180,E1 -490.327,E2 -490.327} C_VEL
LIN {X 0,Y 608.482,Z 176.311,A -85,B 0,C 180,E1 -493.31,E2 -493.31} C_VEL
LIN {X 0,Y 608.445,Z 176.316,A -85,B 0,C 180,E1 -496.128,E2 -496.128} C_VEL
LIN {X 0,Y 608.461,Z 176.319,A -85,B 0,C 180,E1 -498.824,E2 -498.824} C_VEL
LIN {X 0,Y 608.435,Z 176.315,A -85,B 0,C 180,E1 -501.41,E2 -501.41} C_VEL
LIN {X 0,Y 608.437,Z 176.317,A -85,B 0,C 180,E1 -503.955,E2 -503.955} C_VEL
LIN {X 0,Y 608.462,Z 176.32,A -85,B 0,C 180,E1 -506.329,E2 -506.329} C_VEL
LIN {X 0,Y 608.475,Z 176.315,A -85,B 0,C 180,E1 -508.727,E2 -508.727} C_VEL
LIN {X 0,Y 608.454,Z 176.312,A -85,B 0,C 180,E1 -511.382,E2 -511.382} C_VEL
LIN {X 0,Y 608.439,Z 176.319,A -85,B 0,C 180,E1 -513.964,E2 -513.964} C_VEL
LIN {X 0,Y 608.461,Z 176.321,A -85,B 0,C 180,E1 -516.155,E2 -516.155} C_VEL
LIN {X 0,Y 608.447,Z 176.313,A -85,B 0,C 180,E1 -519.018,E2 -519.018} C_VEL
LIN {X 0,Y 608.447,Z 176.319,A -85,B 0,C 180,E1 -521.828,E2 -521.828} C_VEL
LIN {X 0,Y 608.473,Z 176.312,A -85,B 0,C 180,E1 -524.594,E2 -524.594} C_VEL
LIN {X 0,Y 608.464,Z 176.313,A -85,B 0,C 180,E1 -527.323,E2 -527.323} C_VEL
LIN {X 0,Y 608.452,Z 176.32,A -85,B 0,C 180,E1 -530.023,E2 -530.023} C_VEL
LIN {X 0,Y 608.462,Z 176.312,A -85,B 0,C 180,E1 -532.701,E2 -532.701} C_VEL
LIN {X 0,Y 608.445,Z 176.318,A -85,B 0,C 180,E1 -535.362,E2 -535.362} C_VEL
LIN {X 0,Y 608.454,Z 176.317,A -85,B 0,C 180,E1 -538.014,E2 -538.014} C_VEL
LIN {X 0,Y 608.475,Z 176.31,A -85,B 0,C 180,E1 -540.662,E2 -540.662} C_VEL
LIN {X 0,Y 608.473,Z 176.316,A -85,B 0,C 180,E1 -543.311,E2 -543.311} C_VEL
LIN {X 0,Y 608.456,Z 176.315,A -85,B 0,C 180,E1 -545.967,E2 -545.967} C_VEL
LIN {X 0,Y 608.454,Z 176.313,A -85,B 0,C 180,E1 -548.636,E2 -548.636} C_VEL
LIN {X 0,Y 608.456,Z 176.318,A -85,B 0,C 180,E1 -549.461,E2 -549.461} C_VEL
LIN {X 0,Y 607.775,Z 176.399,A -85,B 0,C 180,E1 -550.014,E2 -550.014} C_VEL
LIN {X 0,Y 604.919,Z 176.756,A -85,B 0,C 180,E1 -550.91,E2 -550.91} C_VEL
LIN {X 0,Y 602.517,Z 177.057,A -85,B 0,C 180,E1 -551.632,E2 -551.632} C_VEL
LIN {X 0,Y 601.489,Z 177.18,A -85,B 0,C 180,E1 -552.189,E2 -552.189} C_VEL
LIN {X 0,Y 601.406,Z 177.19,A -85,B 0,C 180,E1 -552.377,E2 -552.377} C_VEL
LIN {X 0,Y 601.426,Z 177.192,A -85,B 0,C 180,E1 -554.897,E2 -554.897} C_VEL
LIN {X 0,Y 601.431,Z 177.193,A -85,B 0,C 180,E1 -556.986,E2 -556.986} C_VEL
LIN {X 0,Y 601.407,Z 177.191,A -85,B 0,C 180,E1 -559.81,E2 -559.81} C_VEL
LIN {X 0,Y 601.409,Z 177.194,A -85,B 0,C 180,E1 -562.683,E2 -562.683} C_VEL
LIN {X 0,Y 601.403,Z 177.198,A -85,B 0,C 180,E1 -564.879,E2 -564.879} C_VEL
LIN {X 0,Y 601.416,Z 177.192,A -85,B 0,C 180,E1 -567.363,E2 -567.363} C_VEL
LIN {X 0,Y 601.427,Z 177.188,A -85,B 0,C 180,E1 -570.164,E2 -570.164} C_VEL
LIN {X 0,Y 601.416,Z 177.197,A -85,B 0,C 180,E1 -572.715,E2 -572.715} C_VEL
LIN {X 0,Y 601.415,Z 177.194,A -85,B 0,C 180,E1 -575.115,E2 -575.115} C_VEL
LIN {X 0,Y 601.432,Z 177.188,A -85,B 0,C 180,E1 -577.419,E2 -577.419} C_VEL
LIN {X 0,Y 601.401,Z 177.191,A -85,B 0,C 180,E1 -579.996,E2 -579.996} C_VEL
LIN {X 0,Y 601.407,Z 177.199,A -85,B 0,C 180,E1 -582.671,E2 -582.671} C_VEL
LIN {X 0,Y 601.426,Z 177.188,A -85,B 0,C 180,E1 -585.482,E2 -585.482} C_VEL
LIN {X 0,Y 601.423,Z 177.198,A -85,B 0,C 180,E1 -588.407,E2 -588.407} C_VEL
LIN {X 0,Y 601.4,Z 177.194,A -85,B 0,C 180,E1 -590.873,E2 -590.873} C_VEL
LIN {X 0,Y 601.397,Z 177.191,A -85,B 0,C 180,E1 -593.417,E2 -593.417} C_VEL
LIN {X 0,Y 601.432,Z 177.194,A -85,B 0,C 180,E1 -596.065,E2 -596.065} C_VEL
LIN {X 0,Y 601.418,Z 177.194,A -85,B 0,C 180,E1 -598.546,E2 -598.546} C_VEL
LIN {X 0,Y 601.429,Z 177.189,A -85,B 0,C 180,E1 -601.373,E2 -601.373} C_VEL
LIN {X 0,Y 601.407,Z 177.2,A -85,B 0,C 180,E1 -604.134,E2 -604.134} C_VEL
LIN {X 0,Y 601.48,Z 177.408,A -85,B 0,C 180,E1 -605.802,E2 -605.802} C_VEL
LIN {X 0,Y 601.77,Z 180.611,A -85,B 0,C 180,E1 -606.239,E2 -606.239} C_VEL
LIN {X 0,Y 601.69,Z 200.879,A -85,B 0,C 180,E1 -608.771,E2 -608.771} C_VEL
LIN {X 0,Y 601.606,Z 224.043,A -85,B 0,C 180,E1 -611.614,E2 -611.614} C_VEL
LIN {X 0,Y 601.545,Z 244.522,A -85,B 0,C 180,E1 -614.064,E2 -614.064} C_VEL
LIN {X 0,Y 601.815,Z 248.487,A -85,B 0,C 180,E1 -614.137,E2 -614.137} C_VEL
LIN {X 0,Y 601.732,Z 382.044,A -85,B 0,C 180,E1 -615.767,E2 -615.767} C_VEL
LIN {X 0,Y 601.712,Z 396.516,A -85,B 0,C 180,E1 -616.081,E2 -616.081} C_VEL
LIN {X 0,Y 601.673,Z 409.533,A -85,B 0,C 180,E1 -616.49,E2 -616.49} C_VEL
LIN {X 0,Y 601.632,Z 421.959,A -85,B 0,C 180,E1 -617.005,E2 -617.005} C_VEL
LIN {X 0,Y 601.561,Z 434.941,A -85,B 0,C 180,E1 -617.689,E2 -617.689} C_VEL
LIN {X 0,Y 601.514,Z 446.699,A -85,B 0,C 180,E1 -618.458,E2 -618.458} C_VEL
LIN {X 0,Y 601.481,Z 458.418,A -85,B 0,C 180,E1 -619.395,E2 -619.395} C_VEL
LIN {X 0,Y 601.431,Z 468.902,A -85,B 0,C 180,E1 -620.414,E2 -620.414} C_VEL
LIN {X 0,Y 601.406,Z 477.553,A -85,B 0,C 180,E1 -621.431,E2 -621.431} C_VEL
LIN {X 0,Y 601.392,Z 485.842,A -85,B 0,C 180,E1 -622.614,E2 -622.614} C_VEL
LIN {X 0,Y 601.361,Z 491.512,A -85,B 0,C 180,E1 -623.605,E2 -623.605} C_VEL
LIN {X 0,Y 601.355,Z 496.376,A -85,B 0,C 180,E1 -624.635,E2 -624.635} C_VEL
LIN {X 0,Y 601.345,Z 501.3,A -85,B 0,C 180,E1 -625.979,E2 -625.979} C_VEL
LIN {X 0,Y 601.324,Z 504.735,A -85,B 0,C 180,E1 -627.32,E2 -627.32} C_VEL
LIN {X 0,Y 601.346,Z 506.779,A -85,B 0,C 180,E1 -628.66,E2 -628.66} C_VEL
LIN {X 0,Y 601.334,Z 507.495,A -85,B 0,C 180,E1 -630,E2 -630} C_VEL
LIN {X 0,Y 601.343,Z 506.883,A -85,B 0,C 180,E1 -631.339,E2 -631.339} C_VEL
LIN {X 0,Y 601.321,Z 504.929,A -85,B 0,C 180,E1 -632.679,E2 -632.679} C_VEL
LIN {X 0,Y 601.346,Z 501.585,A -85,B 0,C 180,E1 -634.021,E2 -634.021} C_VEL
LIN {X 0,Y 601.355,Z 496.759,A -85,B 0,C 180,E1 -635.364,E2 -635.364} C_VEL
LIN {X 0,Y 601.368,Z 490.889,A -85,B 0,C 180,E1 -636.601,E2 -636.601} C_VEL
LIN {X 0,Y 601.386,Z 484.219,A -85,B 0,C 180,E1 -637.723,E2 -637.723} C_VEL
LIN {X 0,Y 601.411,Z 475.562,A -85,B 0,C 180,E1 -638.907,E2 -638.907} C_VEL
LIN {X 0,Y 601.432,Z 466.517,A -85,B 0,C 180,E1 -639.925,E2 -639.925} C_VEL
LIN {X 0,Y 601.474,Z 455.337,A -85,B 0,C 180,E1 -640.963,E2 -640.963} C_VEL
LIN {X 0,Y 601.542,Z 443.107,A -85,B 0,C 180,E1 -641.883,E2 -641.883} C_VEL
LIN {X 0,Y 601.562,Z 430.476,A -85,B 0,C 180,E1 -642.653,E2 -642.653} C_VEL
LIN {X 0,Y 601.63,Z 418.202,A -85,B 0,C 180,E1 -643.253,E2 -643.253} C_VEL
LIN {X 0,Y 601.697,Z 404.167,A -85,B 0,C 180,E1 -643.783,E2 -643.783} C_VEL
LIN {X 0,Y 601.729,Z 390.539,A -85,B 0,C 180,E1 -644.155,E2 -644.155} C_VEL
LIN {X 0,Y 601.728,Z 376.602,A -85,B 0,C 180,E1 -644.401,E2 -644.401} C_VEL
LIN {X 0,Y 601.76,Z 245.871,A -85,B 0,C 180,E1 -645.986,E2 -645.986} C_VEL
LIN {X 0,Y 601.546,Z 244.019,A -85,B 0,C 180,E1 -646.066,E2 -646.066} C_VEL
LIN {X 0,Y 601.618,Z 220.774,A -85,B 0,C 180,E1 -648.874,E2 -648.874} C_VEL
LIN {X 0,Y 601.709,Z 197.264,A -85,B 0,C 180,E1 -651.767,E2 -651.767} C_VEL
LIN {X 0,Y 601.784,Z 179.88,A -85,B 0,C 180,E1 -653.943,E2 -653.943} C_VEL
LIN {X 0,Y 601.466,Z 177.384,A -85,B 0,C 180,E1 -654.298,E2 -654.298} C_VEL
LIN {X 0,Y 601.415,Z 177.19,A -85,B 0,C 180,E1 -657.112,E2 -657.112} C_VEL
LIN {X 0,Y 601.402,Z 177.194,A -85,B 0,C 180,E1 -659.393,E2 -659.393} C_VEL
LIN {X 0,Y 601.401,Z 177.199,A -85,B 0,C 180,E1 -661.726,E2 -661.726} C_VEL
LIN {X 0,Y 601.425,Z 177.193,A -85,B 0,C 180,E1 -664.118,E2 -664.118} C_VEL
LIN {X 0,Y 601.4,Z 177.191,A -85,B 0,C 180,E1 -666.582,E2 -666.582} C_VEL
LIN {X 0,Y 601.403,Z 177.193,A -85,B 0,C 180,E1 -669.126,E2 -669.126} C_VEL
LIN {X 0,Y 601.421,Z 177.196,A -85,B 0,C 180,E1 -671.764,E2 -671.764} C_VEL
LIN {X 0,Y 601.421,Z 177.189,A -85,B 0,C 180,E1 -674.535,E2 -674.535} C_VEL
LIN {X 0,Y 601.409,Z 177.199,A -85,B 0,C 180,E1 -677.408,E2 -677.408} C_VEL
LIN {X 0,Y 601.401,Z 177.192,A -85,B 0,C 180,E1 -680.004,E2 -680.004} C_VEL
LIN {X 0,Y 601.428,Z 177.189,A -85,B 0,C 180,E1 -682.617,E2 -682.617} C_VEL
LIN {X 0,Y 601.436,Z 177.193,A -85,B 0,C 180,E1 -685.069,E2 -685.069} C_VEL
LIN {X 0,Y 601.427,Z 177.194,A -85,B 0,C 180,E1 -687.484,E2 -687.484} C_VEL
LIN {X 0,Y 601.443,Z 177.186,A -85,B 0,C 180,E1 -689.847,E2 -689.847} C_VEL
LIN {X 0,Y 601.447,Z 177.191,A -85,B 0,C 180,E1 -692.889,E2 -692.889} C_VEL
LIN {X 0,Y 601.457,Z 177.184,A -85,B 0,C 180,E1 -695.859,E2 -695.859} C_VEL
LIN {X 0,Y 601.402,Z 177.198,A -85,B 0,C 180,E1 -698.76,E2 -698.76} C_VEL
LIN {X 0,Y 601.416,Z 177.19,A -85,B 0,C 180,E1 -701.608,E2 -701.608} C_VEL
LIN {X 0,Y 601.413,Z 177.193,A -85,B 0,C 180,E1 -704.409,E2 -704.409} C_VEL
LIN {X 0,Y 601.421,Z 177.192,A -85,B 0,C 180,E1 -707.172,E2 -707.172} C_VEL
LIN {X 0,Y 601.428,Z 177.188,A -85,B 0,C 180,E1 -709.905,E2 -709.905} C_VEL
LIN {X 0,Y 601.448,Z 177.195,A -85,B 0,C 180,E1 -712.615,E2 -712.615} C_VEL
LIN {X 0,Y 601.421,Z 177.189,A -85,B 0,C 180,E1 -715.308,E2 -715.308} C_VEL
LIN {X 0,Y 601.421,Z 177.191,A -85,B 0,C 180,E1 -717.991,E2 -717.991} C_VEL
LIN {X 0,Y 601.446,Z 177.191,A -85,B 0,C 180,E1 -720.669,E2 -720.669} C_VEL
LIN {X 0,Y 601.426,Z 177.188,A -85,B 0,C 180,E1 -723.349,E2 -723.349} C_VEL
LIN {X 0,Y 601.409,Z 177.196,A -85,B 0,C 180,E1 -726.037,E2 -726.037} C_VEL
LIN {X 0,Y 601.429,Z 177.19,A -85,B 0,C 180,E1 -728.738,E2 -728.738} C_VEL
LIN {X 0,Y 601.43,Z 177.189,A -85,B 0,C 180,E1 -731.458,E2 -731.458} C_VEL
LIN {X 0,Y 601.411,Z 177.198,A -85,B 0,C 180,E1 -734.206,E2 -734.206} C_VEL
LIN {X 0,Y 601.426,Z 177.188,A -85,B 0,C 180,E1 -736.986,E2 -736.986} C_VEL
LIN {X 0,Y 601.403,Z 177.199,A -85,B 0,C 180,E1 -739.809,E2 -739.809} C_VEL
LIN {X 0,Y 601.404,Z 177.191,A -85,B 0,C 180,E1 -742.683,E2 -742.683} C_VEL
LIN {X 0,Y 601.399,Z 177.191,A -85,B 0,C 180,E1 -744.879,E2 -744.879} C_VEL
LIN {X 0,Y 601.412,Z 177.197,A -85,B 0,C 180,E1 -747.868,E2 -747.868} C_VEL
LIN {X 0,Y 601.397,Z 177.194,A -85,B 0,C 180,E1 -750.166,E2 -750.166} C_VEL
LIN {X 0,Y 601.407,Z 177.189,A -85,B 0,C 180,E1 -752.715,E2 -752.715} C_VEL
LIN {X 0,Y 601.412,Z 177.193,A -85,B 0,C 180,E1 -755.116,E2 -755.116} C_VEL
LIN {X 0,Y 601.429,Z 177.197,A -85,B 0,C 180,E1 -757.419,E2 -757.419} C_VEL
LIN {X 0,Y 601.404,Z 177.193,A -85,B 0,C 180,E1 -759.996,E2 -759.996} C_VEL
LIN {X 0,Y 601.403,Z 177.192,A -85,B 0,C 180,E1 -762.671,E2 -762.671} C_VEL
LIN {X 0,Y 601.392,Z 177.199,A -85,B 0,C 180,E1 -765.48,E2 -765.48} C_VEL
LIN {X 0,Y 601.415,Z 177.19,A -85,B 0,C 180,E1 -768.408,E2 -768.408} C_VEL
LIN {X 0,Y 601.405,Z 177.194,A -85,B 0,C 180,E1 -770.874,E2 -770.874} C_VEL
LIN {X 0,Y 601.398,Z 177.196,A -85,B 0,C 180,E1 -773.418,E2 -773.418} C_VEL
LIN {X 0,Y 601.41,Z 177.19,A -85,B 0,C 180,E1 -776.067,E2 -776.067} C_VEL
LIN {X 0,Y 601.415,Z 177.193,A -85,B 0,C 180,E1 -778.546,E2 -778.546} C_VEL
LIN {X 0,Y 601.403,Z 177.195,A -85,B 0,C 180,E1 -781.372,E2 -781.372} C_VEL
LIN {X 0,Y 601.384,Z 177.198,A -85,B 0,C 180,E1 -783.636,E2 -783.636} C_VEL
LIN {X 0,Y 601.465,Z 177.369,A -85,B 0,C 180,E1 -784.501,E2 -784.501} C_VEL
LIN {X 0,Y 601.983,Z 179.627,A -85,B 0,C 180,E1 -784.779,E2 -784.779} C_VEL
LIN {X 0,Y 601.798,Z 205.886,A -85,B 0,C 180,E1 -787.44,E2 -787.44} C_VEL
LIN {X 0,Y 601.72,Z 231.815,A -85,B 0,C 180,E1 -790.024,E2 -790.024} C_VEL
LIN {X 0,Y 601.727,Z 245.084,A -85,B 0,C 180,E1 -791.308,E2 -791.308} C_VEL
LIN {X 0,Y 602.028,Z 250.015,A -85,B 0,C 180,E1 -791.388,E2 -791.388} C_VEL
LIN {X 0,Y 601.893,Z 412.205,A -85,B 0,C 180,E1 -793.392,E2 -793.392} C_VEL
LIN {X 0,Y 601.835,Z 427.729,A -85,B 0,C 180,E1 -793.725,E2 -793.725} C_VEL
LIN {X 0,Y 601.779,Z 443.06,A -85,B 0,C 180,E1 -794.202,E2 -794.202} C_VEL
LIN {X 0,Y 601.718,Z 456.771,A -85,B 0,C 180,E1 -794.764,E2 -794.764} C_VEL
LIN {X 0,Y 601.664,Z 470.242,A -85,B 0,C 180,E1 -795.455,E2 -795.455} C_VEL
LIN {X 0,Y 601.617,Z 483.454,A -85,B 0,C 180,E1 -796.284,E2 -796.284} C_VEL
LIN {X 0,Y 601.531,Z 495.29,A -85,B 0,C 180,E1 -797.175,E2 -797.175} C_VEL
LIN {X 0,Y 601.487,Z 506.752,A -85,B 0,C 180,E1 -798.202,E2 -798.202} C_VEL
LIN {X 0,Y 601.431,Z 516.392,A -85,B 0,C 180,E1 -799.225,E2 -799.225} C_VEL
LIN {X 0,Y 601.428,Z 525.857,A -85,B 0,C 180,E1 -800.415,E2 -800.415} C_VEL
LIN {X 0,Y 601.369,Z 533.732,A -85,B 0,C 180,E1 -801.6,E2 -801.6} C_VEL
LIN {X 0,Y 601.368,Z 541.089,A -85,B 0,C 180,E1 -802.952,E2 -802.952} C_VEL
LIN {X 0,Y 601.373,Z 546.925,A -85,B 0,C 180,E1 -804.299,E2 -804.299} C_VEL
LIN {X 0,Y 601.33,Z 550.384,A -85,B 0,C 180,E1 -805.308,E2 -805.308} C_VEL
LIN {X 0,Y 601.337,Z 553.887,A -85,B 0,C 180,E1 -806.65,E2 -806.65} C_VEL
LIN {X 0,Y 601.343,Z 556.192,A -85,B 0,C 180,E1 -807.991,E2 -807.991} C_VEL
LIN {X 0,Y 601.337,Z 557.35,A -85,B 0,C 180,E1 -809.331,E2 -809.331} C_VEL
LIN {X 0,Y 601.337,Z 557.35,A -85,B 0,C 180,E1 -810.67,E2 -810.67} C_VEL
LIN {X 0,Y 601.343,Z 556.191,A -85,B 0,C 180,E1 -812.01,E2 -812.01} C_VEL
LIN {X 0,Y 601.337,Z 553.885,A -85,B 0,C 180,E1 -813.35,E2 -813.35} C_VEL
LIN {X 0,Y 601.33,Z 550.383,A -85,B 0,C 180,E1 -814.693,E2 -814.693} C_VEL
LIN {X 0,Y 601.357,Z 545.607,A -85,B 0,C 180,E1 -816.038,E2 -816.038} C_VEL
LIN {X 0,Y 601.366,Z 539.424,A -85,B 0,C 180,E1 -817.386,E2 -817.386} C_VEL
LIN {X 0,Y 601.389,Z 531.652,A -85,B 0,C 180,E1 -818.738,E2 -818.738} C_VEL
LIN {X 0,Y 601.427,Z 523.369,A -85,B 0,C 180,E1 -819.925,E2 -819.925} C_VEL
LIN {X 0,Y 601.461,Z 512.928,A -85,B 0,C 180,E1 -821.165,E2 -821.165} C_VEL
LIN {X 0,Y 601.514,Z 503.191,A -85,B 0,C 180,E1 -822.141,E2 -822.141} C_VEL
LIN {X 0,Y 601.57,Z 491.015,A -85,B 0,C 180,E1 -823.168,E2 -823.168} C_VEL
LIN {X 0,Y 601.606,Z 479.075,A -85,B 0,C 180,E1 -824.012,E2 -824.012} C_VEL
LIN {X 0,Y 601.675,Z 465.525,A -85,B 0,C 180,E1 -824.804,E2 -824.804} C_VEL
LIN {X 0,Y 601.742,Z 450.841,A -85,B 0,C 180,E1 -825.496,E2 -825.496} C_VEL
LIN {X 0,Y 601.795,Z 436.616,A -85,B 0,C 180,E1 -826.016,E2 -826.016} C_VEL
LIN {X 0,Y 601.864,Z 421.583,A -85,B 0,C 180,E1 -826.422,E2 -826.422} C_VEL
LIN {X 0,Y 601.901,Z 406.487,A -85,B 0,C 180,E1 -826.692,E2 -826.692} C_VEL
LIN {X 0,Y 601.96,Z 246.567,A -85,B 0,C 180,E1 -828.656,E2 -828.656} C_VEL
LIN {X 0,Y 601.703,Z 244.698,A -85,B 0,C 180,E1 -828.721,E2 -828.721} C_VEL
LIN {X 0,Y 601.749,Z 219.213,A -85,B 0,C 180,E1 -831.227,E2 -831.227} C_VEL
LIN {X 0,Y 601.929,Z 190.419,A -85,B 0,C 180,E1 -834.12,E2 -834.12} C_VEL
LIN {X 0,Y 601.983,Z 179.622,A -85,B 0,C 180,E1 -835.222,E2 -835.222} C_VEL
LIN {X 0,Y 601.442,Z 177.288,A -85,B 0,C 180,E1 -835.524,E2 -835.524} C_VEL
LIN {X 0,Y 601.385,Z 177.195,A -85,B 0,C 180,E1 -837.869,E2 -837.869} C_VEL
LIN {X 0,Y 601.398,Z 177.184,A -85,B 0,C 180,E1 -840.166,E2 -840.166} C_VEL
LIN {X 0,Y 601.403,Z 177.196,A -85,B 0,C 180,E1 -842.713,E2 -842.713} C_VEL
LIN {X 0,Y 601.392,Z 177.2,A -85,B 0,C 180,E1 -845.111,E2 -845.111} C_VEL
LIN {X 0,Y 601.432,Z 177.19,A -85,B 0,C 180,E1 -847.419,E2 -847.419} C_VEL
LIN {X 0,Y 601.398,Z 177.19,A -85,B 0,C 180,E1 -849.996,E2 -849.996} C_VEL
LIN {X 0,Y 601.405,Z 177.199,A -85,B 0,C 180,E1 -852.67,E2 -852.67} C_VEL
LIN {X 0,Y 601.396,Z 177.192,A -85,B 0,C 180,E1 -855.479,E2 -855.479} C_VEL
LIN {X 0,Y 601.419,Z 177.195,A -85,B 0,C 180,E1 -858.407,E2 -858.407} C_VEL
LIN {X 0,Y 601.427,Z 177.193,A -85,B 0,C 180,E1 -860.875,E2 -860.875} C_VEL
LIN {X 0,Y 601.4,Z 177.191,A -85,B 0,C 180,E1 -863.417,E2 -863.417} C_VEL
LIN {X 0,Y 601.428,Z 177.192,A -85,B 0,C 180,E1 -866.064,E2 -866.064} C_VEL
LIN {X 0,Y 601.417,Z 177.19,A -85,B 0,C 180,E1 -869.058,E2 -869.058} C_VEL
LIN {X 0,Y 601.416,Z 177.189,A -85,B 0,C 180,E1 -871.372,E2 -871.372} C_VEL
LIN {X 0,Y 601.397,Z 177.192,A -85,B 0,C 180,E1 -873.636,E2 -873.636} C_VEL
LIN {X 0,Y 601.415,Z 177.193,A -85,B 0,C 180,E1 -876.59,E2 -876.59} C_VEL
LIN {X 0,Y 601.416,Z 177.19,A -85,B 0,C 180,E1 -879.478,E2 -879.478} C_VEL
LIN {X 0,Y 601.401,Z 177.197,A -85,B 0,C 180,E1 -882.312,E2 -882.312} C_VEL
LIN {X 0,Y 601.422,Z 177.188,A -85,B 0,C 180,E1 -885.103,E2 -885.103} C_VEL
LIN {X 0,Y 601.414,Z 177.199,A -85,B 0,C 180,E1 -887.858,E2 -887.858} C_VEL
LIN {X 0,Y 601.416,Z 177.19,A -85,B 0,C 180,E1 -890.584,E2 -890.584} C_VEL
LIN {X 0,Y 601.428,Z 177.191,A -85,B 0,C 180,E1 -893.344,E2 -893.344} C_VEL
LIN {X 0,Y 601.405,Z 177.197,A -85,B 0,C 180,E1 -895.979,E2 -895.979} C_VEL
LIN {X 0,Y 601.423,Z 177.188,A -85,B 0,C 180,E1 -898.661,E2 -898.661} C_VEL
LIN {X 0,Y 601.416,Z 177.195,A -85,B 0,C 180,E1 -901.339,E2 -901.339} C_VEL
LIN {X 0,Y 601.405,Z 177.193,A -85,B 0,C 180,E1 -904.021,E2 -904.021} C_VEL
LIN {X 0,Y 601.45,Z 177.185,A -85,B 0,C 180,E1 -906.711,E2 -906.711} C_VEL
LIN {X 0,Y 601.413,Z 177.199,A -85,B 0,C 180,E1 -909.459,E2 -909.459} C_VEL
LIN {X 0,Y 601.414,Z 177.19,A -85,B 0,C 180,E1 -912.143,E2 -912.143} C_VEL
LIN {X 0,Y 601.406,Z 177.19,A -85,B 0,C 180,E1 -912.377,E2 -912.377} C_VEL
LIN {X 0,Y 600.743,Z 177.278,A -85,B 0,C 180,E1 -912.936,E2 -912.936} C_VEL
LIN {X 0,Y 597.893,Z 177.634,A -85,B 0,C 180,E1 -913.844,E2 -913.844} C_VEL
LIN {X 0,Y 595.482,Z 177.936,A -85,B 0,C 180,E1 -914.574,E2 -914.574} C_VEL
LIN {X 0,Y 594.444,Z 178.066,A -85,B 0,C 180,E1 -915.138,E2 -915.138} C_VEL
LIN {X 0,Y 594.358,Z 178.072,A -85,B 0,C 180,E1 -915.329,E2 -915.329} C_VEL
LIN {X 0,Y 594.388,Z 178.074,A -85,B 0,C 180,E1 -917.194,E2 -917.194} C_VEL
LIN {X 0,Y 594.374,Z 178.066,A -85,B 0,C 180,E1 -920.054,E2 -920.054} C_VEL
LIN {X 0,Y 594.361,Z 178.077,A -85,B 0,C 180,E1 -922.968,E2 -922.968} C_VEL
LIN {X 0,Y 594.373,Z 178.074,A -85,B 0,C 180,E1 -925.193,E2 -925.193} C_VEL
LIN {X 0,Y 594.384,Z 178.066,A -85,B 0,C 180,E1 -927.527,E2 -927.527} C_VEL
LIN {X 0,Y 594.385,Z 178.066,A -85,B 0,C 180,E1 -930.329,E2 -930.329} C_VEL
LIN {X 0,Y 594.375,Z 178.074,A -85,B 0,C 180,E1 -932.951,E2 -932.951} C_VEL
LIN {X 0,Y 594.383,Z 178.066,A -85,B 0,C 180,E1 -935.407,E2 -935.407} C_VEL
LIN {X 0,Y 594.385,Z 178.066,A -85,B 0,C 180,E1 -937.941,E2 -937.941} C_VEL
LIN {X 0,Y 594.373,Z 178.074,A -85,B 0,C 180,E1 -940.822,E2 -940.822} C_VEL
LIN {X 0,Y 594.365,Z 178.068,A -85,B 0,C 180,E1 -943.3,E2 -943.3} C_VEL
LIN {X 0,Y 594.368,Z 178.072,A -85,B 0,C 180,E1 -946.161,E2 -946.161} C_VEL
LIN {X 0,Y 594.379,Z 178.075,A -85,B 0,C 180,E1 -948.536,E2 -948.536} C_VEL
LIN {X 0,Y 594.372,Z 178.067,A -85,B 0,C 180,E1 -951.297,E2 -951.297} C_VEL
LIN {X 0,Y 594.36,Z 178.07,A -85,B 0,C 180,E1 -953.756,E2 -953.756} C_VEL
LIN {X 0,Y 594.377,Z 178.075,A -85,B 0,C 180,E1 -956.239,E2 -956.239} C_VEL
LIN {X 0,Y 594.368,Z 178.071,A -85,B 0,C 180,E1 -958.65,E2 -958.65} C_VEL
LIN {X 0,Y 594.381,Z 178.067,A -85,B 0,C 180,E1 -961.043,E2 -961.043} C_VEL
LIN {X 0,Y 594.369,Z 178.077,A -85,B 0,C 180,E1 -964.056,E2 -964.056} C_VEL
LIN {X 0,Y 594.432,Z 178.349,A -85,B 0,C 180,E1 -965.62,E2 -965.62} C_VEL
LIN {X 0,Y 594.922,Z 182.063,A -85,B 0,C 180,E1 -966.134,E2 -966.134} C_VEL
LIN {X 0,Y 594.798,Z 202.07,A -85,B 0,C 180,E1 -968.662,E2 -968.662} C_VEL
LIN {X 0,Y 594.67,Z 224.048,A -85,B 0,C 180,E1 -971.392,E2 -971.392} C_VEL
LIN {X 0,Y 594.603,Z 244.544,A -85,B 0,C 180,E1 -973.873,E2 -973.873} C_VEL
LIN {X 0,Y 594.986,Z 248.532,A -85,B 0,C 180,E1 -973.95,E2 -973.95} C_VEL
LIN {X 0,Y 594.851,Z 382.814,A -85,B 0,C 180,E1 -975.612,E2 -975.612} C_VEL
LIN {X 0,Y 594.806,Z 397.282,A -85,B 0,C 180,E1 -975.937,E2 -975.937} C_VEL
LIN {X 0,Y 594.754,Z 411.796,A -85,B 0,C 180,E1 -976.417,E2 -976.417} C_VEL
LIN {X 0,Y 594.644,Z 425.479,A -85,B 0,C 180,E1 -977.023,E2 -977.023} C_VEL
LIN {X 0,Y 594.563,Z 437.775,A -85,B 0,C 180,E1 -977.715,E2 -977.715} C_VEL
LIN {X 0,Y 594.528,Z 450.046,A -85,B 0,C 180,E1 -978.569,E2 -978.569} C_VEL
LIN {X 0,Y 594.449,Z 460.359,A -85,B 0,C 180,E1 -979.441,E2 -979.441} C_VEL
LIN {X 0,Y 594.371,Z 470.459,A -85,B 0,C 180,E1 -980.471,E2 -980.471} C_VEL
LIN {X 0,Y 594.324,Z 478.844,A -85,B 0,C 180,E1 -981.5,E2 -981.5} C_VEL
LIN {X 0,Y 594.303,Z 486.858,A -85,B 0,C 180,E1 -982.696,E2 -982.696} C_VEL
LIN {X 0,Y 594.281,Z 493.313,A -85,B 0,C 180,E1 -983.89,E2 -983.89} C_VEL
LIN {X 0,Y 594.235,Z 499.035,A -85,B 0,C 180,E1 -985.251,E2 -985.251} C_VEL
LIN {X 0,Y 594.259,Z 503.199,A -85,B 0,C 180,E1 -986.61,E2 -986.61} C_VEL
LIN {X 0,Y 594.242,Z 505.928,A -85,B 0,C 180,E1 -987.966,E2 -987.966} C_VEL
LIN {X 0,Y 594.235,Z 507.302,A -85,B 0,C 180,E1 -989.322,E2 -989.322} C_VEL
LIN {X 0,Y 594.236,Z 507.356,A -85,B 0,C 180,E1 -990.677,E2 -990.677} C_VEL
LIN {X 0,Y 594.241,Z 506.075,A -85,B 0,C 180,E1 -992.033,E2 -992.033} C_VEL
LIN {X 0,Y 594.259,Z 503.435,A -85,B 0,C 180,E1 -993.39,E2 -993.39} C_VEL
LIN {X 0,Y 594.236,Z 499.364,A -85,B 0,C 180,E1 -994.749,E2 -994.749} C_VEL
LIN {X 0,Y 594.282,Z 493.741,A -85,B 0,C 180,E1 -996.109,E2 -996.109} C_VEL
LIN {X 0,Y 594.303,Z 487.394,A -85,B 0,C 180,E1 -997.303,E2 -997.303} C_VEL
LIN {X 0,Y 594.324,Z 479.497,A -85,B 0,C 180,E1 -998.5,E2 -998.5} C_VEL
LIN {X 0,Y 594.355,Z 471.242,A -85,B 0,C 180,E1 -999.528,E2 -999.528} C_VEL
LIN {X 0,Y 594.448,Z 461.305,A -85,B 0,C 180,E1 -1000.559,E2 -1000.559} C_VEL
LIN {X 0,Y 594.493,Z 450.169,A -85,B 0,C 180,E1 -1001.512,E2 -1001.512} C_VEL
LIN {X 0,Y 594.581,Z 437.839,A -85,B 0,C 180,E1 -1002.37,E2 -1002.37} C_VEL
LIN {X 0,Y 594.665,Z 425.555,A -85,B 0,C 180,E1 -1003.063,E2 -1003.063} C_VEL
LIN {X 0,Y 594.728,Z 411.888,A -85,B 0,C 180,E1 -1003.67,E2 -1003.67} C_VEL
LIN {X 0,Y 594.807,Z 397.453,A -85,B 0,C 180,E1 -1004.148,E2 -1004.148} C_VEL
LIN {X 0,Y 594.866,Z 382.979,A -85,B 0,C 180,E1 -1004.474,E2 -1004.474} C_VEL
LIN {X 0,Y 594.993,Z 254.101,A -85,B 0,C 180,E1 -1006.071,E2 -1006.071} C_VEL
LIN {X 0,Y 594.804,Z 245.848,A -85,B 0,C 180,E1 -1006.178,E2 -1006.178} C_VEL
LIN {X 0,Y 594.554,Z 244.017,A -85,B 0,C 180,E1 -1006.26,E2 -1006.26} C_VEL
LIN {X 0,Y 594.667,Z 221.539,A -85,B 0,C 180,E1 -1009.008,E2 -1009.008} C_VEL
LIN {X 0,Y 594.815,Z 198.707,A -85,B 0,C 180,E1 -1011.85,E2 -1011.85} C_VEL
LIN {X 0,Y 594.94,Z 181.323,A -85,B 0,C 180,E1 -1014.05,E2 -1014.05} C_VEL
LIN {X 0,Y 594.419,Z 178.266,A -85,B 0,C 180,E1 -1014.491,E2 -1014.491} C_VEL
LIN {X 0,Y 594.366,Z 178.069,A -85,B 0,C 180,E1 -1016.7,E2 -1016.7} C_VEL
LIN {X 0,Y 594.376,Z 178.067,A -85,B 0,C 180,E1 -1018.998,E2 -1018.998} C_VEL
LIN {X 0,Y 594.375,Z 178.073,A -85,B 0,C 180,E1 -1021.642,E2 -1021.642} C_VEL
LIN {X 0,Y 594.373,Z 178.067,A -85,B 0,C 180,E1 -1024.58,E2 -1024.58} C_VEL
LIN {X 0,Y 594.378,Z 178.067,A -85,B 0,C 180,E1 -1027.086,E2 -1027.086} C_VEL
LIN {X 0,Y 594.356,Z 178.078,A -85,B 0,C 180,E1 -1029.772,E2 -1029.772} C_VEL
LIN {X 0,Y 594.367,Z 178.067,A -85,B 0,C 180,E1 -1032.375,E2 -1032.375} C_VEL
LIN {X 0,Y 594.36,Z 178.073,A -85,B 0,C 180,E1 -1035.191,E2 -1035.191} C_VEL
LIN {X 0,Y 594.379,Z 178.067,A -85,B 0,C 180,E1 -1038.151,E2 -1038.151} C_VEL
LIN {X 0,Y 594.371,Z 178.066,A -85,B 0,C 180,E1 -1040.319,E2 -1040.319} C_VEL
LIN {X 0,Y 594.379,Z 178.07,A -85,B 0,C 180,E1 -1042.913,E2 -1042.913} C_VEL
LIN {X 0,Y 594.381,Z 178.067,A -85,B 0,C 180,E1 -1045.86,E2 -1045.86} C_VEL
LIN {X 0,Y 594.374,Z 178.069,A -85,B 0,C 180,E1 -1048.65,E2 -1048.65} C_VEL
LIN {X 0,Y 594.379,Z 178.074,A -85,B 0,C 180,E1 -1051.041,E2 -1051.041} C_VEL
LIN {X 0,Y 594.379,Z 178.066,A -85,B 0,C 180,E1 -1053.977,E2 -1053.977} C_VEL
LIN {X 0,Y 594.387,Z 178.065,A -85,B 0,C 180,E1 -1056.296,E2 -1056.296} C_VEL
LIN {X 0,Y 594.398,Z 178.068,A -85,B 0,C 180,E1 -1059.224,E2 -1059.224} C_VEL
LIN {X 0,Y 594.375,Z 178.067,A -85,B 0,C 180,E1 -1062.096,E2 -1062.096} C_VEL
LIN {X 0,Y 594.365,Z 178.069,A -85,B 0,C 180,E1 -1064.219,E2 -1064.219} C_VEL
LIN {X 0,Y 594.369,Z 178.072,A -85,B 0,C 180,E1 -1067.017,E2 -1067.017} C_VEL
LIN {X 0,Y 594.387,Z 178.065,A -85,B 0,C 180,E1 -1069.784,E2 -1069.784} C_VEL
LIN {X 0,Y 594.396,Z 178.073,A -85,B 0,C 180,E1 -1072.527,E2 -1072.527} C_VEL
LIN {X 0,Y 594.39,Z 178.065,A -85,B 0,C 180,E1 -1075.252,E2 -1075.252} C_VEL
LIN {X 0,Y 594.391,Z 178.067,A -85,B 0,C 180,E1 -1077.967,E2 -1077.967} C_VEL
LIN {X 0,Y 594.416,Z 178.066,A -85,B 0,C 180,E1 -1080.677,E2 -1080.677} C_VEL
LIN {X 0,Y 594.378,Z 178.066,A -85,B 0,C 180,E1 -1083.389,E2 -1083.389} C_VEL
LIN {X 0,Y 594.365,Z 178.075,A -85,B 0,C 180,E1 -1086.109,E2 -1086.109} C_VEL
LIN {X 0,Y 594.391,Z 178.065,A -85,B 0,C 180,E1 -1088.842,E2 -1088.842} C_VEL
LIN {X 0,Y 594.388,Z 178.067,A -85,B 0,C 180,E1 -1091.596,E2 -1091.596} C_VEL
LIN {X 0,Y 594.381,Z 178.07,A -85,B 0,C 180,E1 -1094.377,E2 -1094.377} C_VEL
LIN {X 0,Y 594.386,Z 178.065,A -85,B 0,C 180,E1 -1097.193,E2 -1097.193} C_VEL
LIN {X 0,Y 594.368,Z 178.075,A -85,B 0,C 180,E1 -1100.054,E2 -1100.054} C_VEL
LIN {X 0,Y 594.357,Z 178.069,A -85,B 0,C 180,E1 -1102.967,E2 -1102.967} C_VEL
LIN {X 0,Y 594.375,Z 178.068,A -85,B 0,C 180,E1 -1105.193,E2 -1105.193} C_VEL
LIN {X 0,Y 594.378,Z 178.071,A -85,B 0,C 180,E1 -1107.527,E2 -1107.527} C_VEL
LIN {X 0,Y 594.365,Z 178.069,A -85,B 0,C 180,E1 -1110.326,E2 -1110.326} C_VEL
LIN {X 0,Y 594.37,Z 178.067,A -85,B 0,C 180,E1 -1112.951,E2 -1112.951} C_VEL
LIN {X 0,Y 594.373,Z 178.075,A -85,B 0,C 180,E1 -1115.407,E2 -1115.407} C_VEL
LIN {X 0,Y 594.373,Z 178.069,A -85,B 0,C 180,E1 -1117.942,E2 -1117.942} C_VEL
LIN {X 0,Y 594.372,Z 178.069,A -85,B 0,C 180,E1 -1120.823,E2 -1120.823} C_VEL
LIN {X 0,Y 594.36,Z 178.078,A -85,B 0,C 180,E1 -1123.3,E2 -1123.3} C_VEL
LIN {X 0,Y 594.354,Z 178.069,A -85,B 0,C 180,E1 -1126.162,E2 -1126.162} C_VEL
LIN {X 0,Y 594.371,Z 178.075,A -85,B 0,C 180,E1 -1129.179,E2 -1129.179} C_VEL
LIN {X 0,Y 594.37,Z 178.067,A -85,B 0,C 180,E1 -1132.059,E2 -1132.059} C_VEL
LIN {X 0,Y 594.348,Z 178.073,A -85,B 0,C 180,E1 -1134.677,E2 -1134.677} C_VEL
LIN {X 0,Y 594.37,Z 178.075,A -85,B 0,C 180,E1 -1137.09,E2 -1137.09} C_VEL
LIN {X 0,Y 594.361,Z 178.061,A -85,B 0,C 180,E1 -1139.676,E2 -1139.676} C_VEL
LIN {X 0,Y 594.372,Z 178.074,A -85,B 0,C 180,E1 -1142.54,E2 -1142.54} C_VEL
LIN {X 0,Y 594.403,Z 178.26,A -85,B 0,C 180,E1 -1144.27,E2 -1144.27} C_VEL
LIN {X 0,Y 595.178,Z 181.427,A -85,B 0,C 180,E1 -1144.657,E2 -1144.657} C_VEL
LIN {X 0,Y 595.03,Z 203.022,A -85,B 0,C 180,E1 -1146.877,E2 -1146.877} C_VEL
LIN {X 0,Y 594.883,Z 228.216,A -85,B 0,C 180,E1 -1149.423,E2 -1149.423} C_VEL
LIN {X 0,Y 594.835,Z 245.024,A -85,B 0,C 180,E1 -1151.08,E2 -1151.08} C_VEL
LIN {X 0,Y 595.318,Z 248.692,A -85,B 0,C 180,E1 -1151.154,E2 -1151.154} C_VEL
LIN {X 0,Y 595.104,Z 411.932,A -85,B 0,C 180,E1 -1153.192,E2 -1153.192} C_VEL
LIN {X 0,Y 595.027,Z 427.727,A -85,B 0,C 180,E1 -1153.533,E2 -1153.533} C_VEL
LIN {X 0,Y 594.947,Z 443.058,A -85,B 0,C 180,E1 -1154.015,E2 -1154.015} C_VEL
LIN {X 0,Y 594.847,Z 456.774,A -85,B 0,C 180,E1 -1154.584,E2 -1154.584} C_VEL
LIN {X 0,Y 594.74,Z 470.245,A -85,B 0,C 180,E1 -1155.282,E2 -1155.282} C_VEL
LIN {X 0,Y 594.68,Z 482.8,A -85,B 0,C 180,E1 -1156.076,E2 -1156.076} C_VEL
LIN {X 0,Y 594.559,Z 495.292,A -85,B 0,C 180,E1 -1157.022,E2 -1157.022} C_VEL
LIN {X 0,Y 594.465,Z 506.753,A -85,B 0,C 180,E1 -1158.06,E2 -1158.06} C_VEL
LIN {X 0,Y 594.388,Z 516.393,A -85,B 0,C 180,E1 -1159.095,E2 -1159.095} C_VEL
LIN {X 0,Y 594.366,Z 525.858,A -85,B 0,C 180,E1 -1160.3,E2 -1160.3} C_VEL
LIN {X 0,Y 594.312,Z 533.733,A -85,B 0,C 180,E1 -1161.5,E2 -1161.5} C_VEL
LIN {X 0,Y 594.292,Z 541.09,A -85,B 0,C 180,E1 -1162.867,E2 -1162.867} C_VEL
LIN {X 0,Y 594.299,Z 546.925,A -85,B 0,C 180,E1 -1164.231,E2 -1164.231} C_VEL
LIN {X 0,Y 594.232,Z 550.385,A -85,B 0,C 180,E1 -1165.251,E2 -1165.251} C_VEL
LIN {X 0,Y 594.256,Z 553.888,A -85,B 0,C 180,E1 -1166.61,E2 -1166.61} C_VEL
LIN {X 0,Y 594.241,Z 556.193,A -85,B 0,C 180,E1 -1167.967,E2 -1167.967} C_VEL
LIN {X 0,Y 594.237,Z 557.35,A -85,B 0,C 180,E1 -1169.323,E2 -1169.323} C_VEL
LIN {X 0,Y 594.237,Z 557.35,A -85,B 0,C 180,E1 -1170.678,E2 -1170.678} C_VEL
LIN {X 0,Y 594.241,Z 556.192,A -85,B 0,C 180,E1 -1172.034,E2 -1172.034} C_VEL
LIN {X 0,Y 594.256,Z 553.886,A -85,B 0,C 180,E1 -1173.39,E2 -1173.39} C_VEL
LIN {X 0,Y 594.232,Z 550.383,A -85,B 0,C 180,E1 -1174.749,E2 -1174.749} C_VEL
LIN {X 0,Y 594.279,Z 545.607,A -85,B 0,C 180,E1 -1176.11,E2 -1176.11} C_VEL
LIN {X 0,Y 594.287,Z 539.424,A -85,B 0,C 180,E1 -1177.475,E2 -1177.475} C_VEL
LIN {X 0,Y 594.331,Z 531.651,A -85,B 0,C 180,E1 -1178.843,E2 -1178.843} C_VEL
LIN {X 0,Y 594.387,Z 523.369,A -85,B 0,C 180,E1 -1180.044,E2 -1180.044} C_VEL
LIN {X 0,Y 594.434,Z 513.555,A -85,B 0,C 180,E1 -1181.232,E2 -1181.232} C_VEL
LIN {X 0,Y 594.531,Z 503.19,A -85,B 0,C 180,E1 -1182.285,E2 -1182.285} C_VEL
LIN {X 0,Y 594.581,Z 491.016,A -85,B 0,C 180,E1 -1183.326,E2 -1183.326} C_VEL
LIN {X 0,Y 594.694,Z 479.072,A -85,B 0,C 180,E1 -1184.178,E2 -1184.178} C_VEL
LIN {X 0,Y 594.775,Z 465.522,A -85,B 0,C 180,E1 -1184.98,E2 -1184.98} C_VEL
LIN {X 0,Y 594.883,Z 450.837,A -85,B 0,C 180,E1 -1185.679,E2 -1185.679} C_VEL
LIN {X 0,Y 594.973,Z 436.616,A -85,B 0,C 180,E1 -1186.204,E2 -1186.204} C_VEL
LIN {X 0,Y 595.054,Z 422.036,A -85,B 0,C 180,E1 -1186.605,E2 -1186.605} C_VEL
LIN {X 0,Y 595.085,Z 406.487,A -85,B 0,C 180,E1 -1186.889,E2 -1186.889} C_VEL
LIN {X 0,Y 595.317,Z 248.499,A -85,B 0,C 180,E1 -1188.848,E2 -1188.848} C_VEL
LIN {X 0,Y 594.816,Z 244.808,A -85,B 0,C 180,E1 -1188.937,E2 -1188.937} C_VEL
LIN {X 0,Y 594.989,Z 215.613,A -85,B 0,C 180,E1 -1191.844,E2 -1191.844} C_VEL
LIN {X 0,Y 595.18,Z 186.596,A -85,B 0,C 180,E1 -1194.807,E2 -1194.807} C_VEL
LIN {X 0,Y 595.179,Z 181.421,A -85,B 0,C 180,E1 -1195.344,E2 -1195.344} C_VEL
LIN {X 0,Y 594.393,Z 178.174,A -85,B 0,C 180,E1 -1195.755,E2 -1195.755} C_VEL
LIN {X 0,Y 594.354,Z 178.071,A -85,B 0,C 180,E1 -1198.228,E2 -1198.228} C_VEL
LIN {X 0,Y 594.363,Z 178.059,A -85,B 0,C 180,E1 -1200.56,E2 -1200.56} C_VEL
LIN {X 0,Y 594.372,Z 178.075,A -85,B 0,C 180,E1 -1202.95,E2 -1202.95} C_VEL
LIN {X 0,Y 594.346,Z 178.072,A -85,B 0,C 180,E1 -1205.409,E2 -1205.409} C_VEL
LIN {X 0,Y 594.371,Z 178.067,A -85,B 0,C 180,E1 -1207.942,E2 -1207.942} C_VEL
LIN {X 0,Y 594.373,Z 178.074,A -85,B 0,C 180,E1 -1210.822,E2 -1210.822} C_VEL
LIN {X 0,Y 594.357,Z 178.069,A -85,B 0,C 180,E1 -1213.838,E2 -1213.838} C_VEL
LIN {X 0,Y 594.363,Z 178.078,A -85,B 0,C 180,E1 -1216.7,E2 -1216.7} C_VEL
LIN {X 0,Y 594.358,Z 178.069,A -85,B 0,C 180,E1 -1219.432,E2 -1219.432} C_VEL
LIN {X 0,Y 594.384,Z 178.073,A -85,B 0,C 180,E1 -1222.392,E2 -1222.392} C_VEL
LIN {X 0,Y 594.391,Z 178.064,A -85,B 0,C 180,E1 -1225.421,E2 -1225.421} C_VEL
LIN {X 0,Y 594.386,Z 178.073,A -85,B 0,C 180,E1 -1228.355,E2 -1228.355} C_VEL
LIN {X 0,Y 594.377,Z 178.067,A -85,B 0,C 180,E1 -1231.042,E2 -1231.042} C_VEL
LIN {X 0,Y 594.386,Z 178.069,A -85,B 0,C 180,E1 -1233.976,E2 -1233.976} C_VEL
LIN {X 0,Y 594.383,Z 178.074,A -85,B 0,C 180,E1 -1236.296,E2 -1236.296} C_VEL
LIN {X 0,Y 594.39,Z 178.064,A -85,B 0,C 180,E1 -1239.224,E2 -1239.224} C_VEL
LIN {X 0,Y 594.378,Z 178.076,A -85,B 0,C 180,E1 -1242.096,E2 -1242.096} C_VEL
LIN {X 0,Y 594.369,Z 178.067,A -85,B 0,C 180,E1 -1244.922,E2 -1244.922} C_VEL
LIN {X 0,Y 594.387,Z 178.071,A -85,B 0,C 180,E1 -1247.712,E2 -1247.712} C_VEL
LIN {X 0,Y 594.368,Z 178.069,A -85,B 0,C 180,E1 -1250.471,E2 -1250.471} C_VEL
LIN {X 0,Y 594.391,Z 178.065,A -85,B 0,C 180,E1 -1252.527,E2 -1252.527} C_VEL
LIN {X 0,Y 594.385,Z 178.067,A -85,B 0,C 180,E1 -1255.252,E2 -1255.252} C_VEL
LIN {X 0,Y 594.393,Z 178.069,A -85,B 0,C 180,E1 -1257.967,E2 -1257.967} C_VEL
LIN {X 0,Y 594.417,Z 178.061,A -85,B 0,C 180,E1 -1260.678,E2 -1260.678} C_VEL
LIN {X 0,Y 594.376,Z 178.073,A -85,B 0,C 180,E1 -1263.389,E2 -1263.389} C_VEL
LIN {X 0,Y 594.366,Z 178.069,A -85,B 0,C 180,E1 -1266.109,E2 -1266.109} C_VEL
LIN {X 0,Y 594.395,Z 178.065,A -85,B 0,C 180,E1 -1268.842,E2 -1268.842} C_VEL
LIN {X 0,Y 594.391,Z 178.07,A -85,B 0,C 180,E1 -1271.596,E2 -1271.596} C_VEL
LIN {X 0,Y 594.387,Z 178.065,A -85,B 0,C 180,E1 -1274.377,E2 -1274.377} C_VEL
LIN {X 0,Y 594.358,Z 178.072,A -85,B 0,C 180,E1 -1275.329,E2 -1275.329} C_VEL
LIN {X 0,Y 593.685,Z 178.154,A -85,B 0,C 180,E1 -1275.895,E2 -1275.895} C_VEL
LIN {X 0,Y 590.819,Z 178.512,A -85,B 0,C 180,E1 -1276.813,E2 -1276.813} C_VEL
LIN {X 0,Y 588.408,Z 178.814,A -85,B 0,C 180,E1 -1277.551,E2 -1277.551} C_VEL
LIN {X 0,Y 587.385,Z 178.938,A -85,B 0,C 180,E1 -1278.122,E2 -1278.122} C_VEL
LIN {X 0,Y 587.307,Z 178.947,A -85,B 0,C 180,E1 -1278.315,E2 -1278.315} C_VEL
LIN {X 0,Y 587.328,Z 178.952,A -85,B 0,C 180,E1 -1281.038,E2 -1281.038} C_VEL
LIN {X 0,Y 587.32,Z 178.952,A -85,B 0,C 180,E1 -1283.259,E2 -1283.259} C_VEL
LIN {X 0,Y 587.331,Z 178.947,A -85,B 0,C 180,E1 -1285.517,E2 -1285.517} C_VEL
LIN {X 0,Y 587.345,Z 178.941,A -85,B 0,C 180,E1 -1287.818,E2 -1287.818} C_VEL
LIN {X 0,Y 587.335,Z 178.946,A -85,B 0,C 180,E1 -1290.51,E2 -1290.51} C_VEL
LIN {X 0,Y 587.331,Z 178.945,A -85,B 0,C 180,E1 -1293.397,E2 -1293.397} C_VEL
LIN {X 0,Y 587.356,Z 178.94,A -85,B 0,C 180,E1 -1295.896,E2 -1295.896} C_VEL
LIN {X 0,Y 587.328,Z 178.951,A -85,B 0,C 180,E1 -1298.48,E2 -1298.48} C_VEL
LIN {X 0,Y 587.333,Z 178.946,A -85,B 0,C 180,E1 -1301.157,E2 -1301.157} C_VEL
LIN {X 0,Y 587.311,Z 178.949,A -85,B 0,C 180,E1 -1304.112,E2 -1304.112} C_VEL
LIN {X 0,Y 587.313,Z 178.948,A -85,B 0,C 180,E1 -1306.994,E2 -1306.994} C_VEL
LIN {X 0,Y 587.311,Z 178.948,A -85,B 0,C 180,E1 -1309.746,E2 -1309.746} C_VEL
LIN {X 0,Y 587.342,Z 178.952,A -85,B 0,C 180,E1 -1312.392,E2 -1312.392} C_VEL
LIN {X 0,Y 587.324,Z 178.946,A -85,B 0,C 180,E1 -1314.944,E2 -1314.944} C_VEL
LIN {X 0,Y 587.34,Z 178.942,A -85,B 0,C 180,E1 -1317.421,E2 -1317.421} C_VEL
LIN {X 0,Y 587.333,Z 178.948,A -85,B 0,C 180,E1 -1319.83,E2 -1319.83} C_VEL
LIN {X 0,Y 587.304,Z 178.953,A -85,B 0,C 180,E1 -1322.316,E2 -1322.316} C_VEL
LIN {X 0,Y 587.326,Z 178.95,A -85,B 0,C 180,E1 -1324.483,E2 -1324.483} C_VEL
LIN {X 0,Y 587.366,Z 179.074,A -85,B 0,C 180,E1 -1325.369,E2 -1325.369} C_VEL
LIN {X 0,Y 588.077,Z 183.516,A -85,B 0,C 180,E1 -1326.026,E2 -1326.026} C_VEL
LIN {X 0,Y 587.902,Z 203.644,A -85,B 0,C 180,E1 -1328.599,E2 -1328.599} C_VEL
LIN {X 0,Y 587.709,Z 226.949,A -85,B 0,C 180,E1 -1331.525,E2 -1331.525} C_VEL
LIN {X 0,Y 587.623,Z 244.575,A -85,B 0,C 180,E1 -1333.676,E2 -1333.676} C_VEL
LIN {X 0,Y 588.182,Z 248.577,A -85,B 0,C 180,E1 -1333.759,E2 -1333.759} C_VEL
LIN {X 0,Y 587.997,Z 382.843,A -85,B 0,C 180,E1 -1335.441,E2 -1335.441} C_VEL
LIN {X 0,Y 587.918,Z 397.133,A -85,B 0,C 180,E1 -1335.764,E2 -1335.764} C_VEL
LIN {X 0,Y 587.856,Z 410.687,A -85,B 0,C 180,E1 -1336.21,E2 -1336.21} C_VEL
LIN {X 0,Y 587.733,Z 423.743,A -85,B 0,C 180,E1 -1336.78,E2 -1336.78} C_VEL
LIN {X 0,Y 587.626,Z 436.375,A -85,B 0,C 180,E1 -1337.48,E2 -1337.48} C_VEL
LIN {X 0,Y 587.514,Z 447.88,A -85,B 0,C 180,E1 -1338.266,E2 -1338.266} C_VEL
LIN {X 0,Y 587.467,Z 458.433,A -85,B 0,C 180,E1 -1339.139,E2 -1339.139} C_VEL
LIN {X 0,Y 587.355,Z 468.912,A -85,B 0,C 180,E1 -1340.183,E2 -1340.183} C_VEL
LIN {X 0,Y 587.311,Z 477.561,A -85,B 0,C 180,E1 -1341.224,E2 -1341.224} C_VEL
LIN {X 0,Y 587.25,Z 485.849,A -85,B 0,C 180,E1 -1342.435,E2 -1342.435} C_VEL
LIN {X 0,Y 587.181,Z 492.472,A -85,B 0,C 180,E1 -1343.636,E2 -1343.636} C_VEL
LIN {X 0,Y 587.158,Z 497.793,A -85,B 0,C 180,E1 -1344.849,E2 -1344.849} C_VEL
LIN {X 0,Y 587.181,Z 501.305,A -85,B 0,C 180,E1 -1345.882,E2 -1345.882} C_VEL
LIN {X 0,Y 587.13,Z 504.739,A -85,B 0,C 180,E1 -1347.255,E2 -1347.255} C_VEL
LIN {X 0,Y 587.145,Z 506.782,A -85,B 0,C 180,E1 -1348.628,E2 -1348.628} C_VEL
LIN {X 0,Y 587.136,Z 507.496,A -85,B 0,C 180,E1 -1350,E2 -1350} C_VEL
LIN {X 0,Y 587.142,Z 506.882,A -85,B 0,C 180,E1 -1351.372,E2 -1351.372} C_VEL
LIN {X 0,Y 587.128,Z 504.928,A -85,B 0,C 180,E1 -1352.744,E2 -1352.744} C_VEL
LIN {X 0,Y 587.182,Z 501.583,A -85,B 0,C 180,E1 -1354.118,E2 -1354.118} C_VEL
LIN {X 0,Y 587.2,Z 496.755,A -85,B 0,C 180,E1 -1355.494,E2 -1355.494} C_VEL
LIN {X 0,Y 587.21,Z 490.291,A -85,B 0,C 180,E1 -1356.874,E2 -1356.874} C_VEL
LIN {X 0,Y 587.269,Z 483.092,A -85,B 0,C 180,E1 -1358.083,E2 -1358.083} C_VEL
LIN {X 0,Y 587.332,Z 475.554,A -85,B 0,C 180,E1 -1359.122,E2 -1359.122} C_VEL
LIN {X 0,Y 587.376,Z 466.506,A -85,B 0,C 180,E1 -1360.165,E2 -1360.165} C_VEL
LIN {X 0,Y 587.503,Z 455.548,A -85,B 0,C 180,E1 -1361.208,E2 -1361.208} C_VEL
LIN {X 0,Y 587.566,Z 444.374,A -85,B 0,C 180,E1 -1362.082,E2 -1362.082} C_VEL
LIN {X 0,Y 587.643,Z 432.03,A -85,B 0,C 180,E1 -1362.87,E2 -1362.87} C_VEL
LIN {X 0,Y 587.783,Z 420.154,A -85,B 0,C 180,E1 -1363.483,E2 -1363.483} C_VEL
LIN {X 0,Y 587.895,Z 406.809,A -85,B 0,C 180,E1 -1364.022,E2 -1364.022} C_VEL
LIN {X 0,Y 587.947,Z 392.809,A -85,B 0,C 180,E1 -1364.438,E2 -1364.438} C_VEL
LIN {X 0,Y 587.992,Z 378.711,A -85,B 0,C 180,E1 -1364.713,E2 -1364.713} C_VEL
LIN {X 0,Y 588.09,Z 247.346,A -85,B 0,C 180,E1 -1366.349,E2 -1366.349} C_VEL
LIN {X 0,Y 587.624,Z 244.278,A -85,B 0,C 180,E1 -1366.435,E2 -1366.435} C_VEL
LIN {X 0,Y 587.745,Z 221.12,A -85,B 0,C 180,E1 -1369.293,E2 -1369.293} C_VEL
LIN {X 0,Y 587.916,Z 200.151,A -85,B 0,C 180,E1 -1371.935,E2 -1371.935} C_VEL
LIN {X 0,Y 588.09,Z 182.935,A -85,B 0,C 180,E1 -1374.139,E2 -1374.139} C_VEL
LIN {X 0,Y 587.336,Z 179.064,A -85,B 0,C 180,E1 -1374.727,E2 -1374.727} C_VEL
LIN {X 0,Y 587.313,Z 178.948,A -85,B 0,C 180,E1 -1377.046,E2 -1377.046} C_VEL
LIN {X 0,Y 587.342,Z 178.946,A -85,B 0,C 180,E1 -1379.379,E2 -1379.379} C_VEL
LIN {X 0,Y 587.343,Z 178.953,A -85,B 0,C 180,E1 -1381.835,E2 -1381.835} C_VEL
LIN {X 0,Y 587.344,Z 178.945,A -85,B 0,C 180,E1 -1384.347,E2 -1384.347} C_VEL
LIN {X 0,Y 587.349,Z 178.941,A -85,B 0,C 180,E1 -1386.746,E2 -1386.746} C_VEL
LIN {X 0,Y 587.329,Z 178.949,A -85,B 0,C 180,E1 -1389.36,E2 -1389.36} C_VEL
LIN {X 0,Y 587.332,Z 178.946,A -85,B 0,C 180,E1 -1392.107,E2 -1392.107} C_VEL
LIN {X 0,Y 587.312,Z 178.95,A -85,B 0,C 180,E1 -1395.088,E2 -1395.088} C_VEL
LIN {X 0,Y 587.349,Z 178.945,A -85,B 0,C 180,E1 -1397.927,E2 -1397.927} C_VEL
LIN {X 0,Y 587.32,Z 178.949,A -85,B 0,C 180,E1 -1401.059,E2 -1401.059} C_VEL
LIN {X 0,Y 587.349,Z 178.952,A -85,B 0,C 180,E1 -1403.291,E2 -1403.291} C_VEL
LIN {X 0,Y 587.363,Z 178.941,A -85,B 0,C 180,E1 -1405.78,E2 -1405.78} C_VEL
LIN {X 0,Y 587.341,Z 178.943,A -85,B 0,C 180,E1 -1408.231,E2 -1408.231} C_VEL
LIN {X 0,Y 587.345,Z 178.947,A -85,B 0,C 180,E1 -1410.866,E2 -1410.866} C_VEL
LIN {X 0,Y 587.353,Z 178.942,A -85,B 0,C 180,E1 -1413.818,E2 -1413.818} C_VEL
LIN {X 0,Y 587.333,Z 178.943,A -85,B 0,C 180,E1 -1415.993,E2 -1415.993} C_VEL
LIN {X 0,Y 587.317,Z 178.946,A -85,B 0,C 180,E1 -1418.225,E2 -1418.225} C_VEL
LIN {X 0,Y 587.344,Z 178.948,A -85,B 0,C 180,E1 -1421.151,E2 -1421.151} C_VEL
LIN {X 0,Y 587.347,Z 178.944,A -85,B 0,C 180,E1 -1423.311,E2 -1423.311} C_VEL
LIN {X 0,Y 587.356,Z 178.943,A -85,B 0,C 180,E1 -1426.154,E2 -1426.154} C_VEL
LIN {X 0,Y 587.337,Z 178.949,A -85,B 0,C 180,E1 -1428.962,E2 -1428.962} C_VEL
LIN {X 0,Y 587.364,Z 178.94,A -85,B 0,C 180,E1 -1431.745,E2 -1431.745} C_VEL
LIN {X 0,Y 587.354,Z 178.951,A -85,B 0,C 180,E1 -1434.507,E2 -1434.507} C_VEL
LIN {X 0,Y 587.372,Z 178.939,A -85,B 0,C 180,E1 -1437.257,E2 -1437.257} C_VEL
LIN {X 0,Y 587.376,Z 178.942,A -85,B 0,C 180,E1 -1440,E2 -1440} C_VEL
LIN {X 0,Y 587.368,Z 178.943,A -85,B 0,C 180,E1 -1442.743,E2 -1442.743} C_VEL
LIN {X 0,Y 587.355,Z 178.941,A -85,B 0,C 180,E1 -1445.493,E2 -1445.493} C_VEL
LIN {X 0,Y 587.364,Z 178.949,A -85,B 0,C 180,E1 -1448.255,E2 -1448.255} C_VEL
LIN {X 0,Y 587.339,Z 178.943,A -85,B 0,C 180,E1 -1451.134,E2 -1451.134} C_VEL
LIN {X 0,Y 587.357,Z 178.947,A -85,B 0,C 180,E1 -1454.261,E2 -1454.261} C_VEL
LIN {X 0,Y 587.353,Z 178.943,A -85,B 0,C 180,E1 -1457.406,E2 -1457.406} C_VEL
LIN {X 0,Y 587.32,Z 178.949,A -85,B 0,C 180,E1 -1460.305,E2 -1460.305} C_VEL
LIN {X 0,Y 587.315,Z 178.948,A -85,B 0,C 180,E1 -1463.259,E2 -1463.259} C_VEL
LIN {X 0,Y 587.333,Z 178.949,A -85,B 0,C 180,E1 -1465.517,E2 -1465.517} C_VEL
LIN {X 0,Y 587.34,Z 178.951,A -85,B 0,C 180,E1 -1467.818,E2 -1467.818} C_VEL
LIN {X 0,Y 587.325,Z 178.945,A -85,B 0,C 180,E1 -1470.51,E2 -1470.51} C_VEL
LIN {X 0,Y 587.332,Z 178.945,A -85,B 0,C 180,E1 -1473.112,E2 -1473.112} C_VEL
LIN {X 0,Y 587.337,Z 178.953,A -85,B 0,C 180,E1 -1475.545,E2 -1475.545} C_VEL
LIN {X 0,Y 587.323,Z 178.944,A -85,B 0,C 180,E1 -1478.48,E2 -1478.48} C_VEL
LIN {X 0,Y 587.331,Z 178.95,A -85,B 0,C 180,E1 -1481.157,E2 -1481.157} C_VEL
LIN {X 0,Y 587.305,Z 178.948,A -85,B 0,C 180,E1 -1484.112,E2 -1484.112} C_VEL
LIN {X 0,Y 587.308,Z 178.953,A -85,B 0,C 180,E1 -1486.994,E2 -1486.994} C_VEL
LIN {X 0,Y 587.303,Z 178.945,A -85,B 0,C 180,E1 -1489.746,E2 -1489.746} C_VEL
LIN {X 0,Y 587.337,Z 178.944,A -85,B 0,C 180,E1 -1492.393,E2 -1492.393} C_VEL
LIN {X 0,Y 587.334,Z 178.945,A -85,B 0,C 180,E1 -1495.654,E2 -1495.654} C_VEL
LIN {X 0,Y 587.327,Z 178.944,A -85,B 0,C 180,E1 -1498.231,E2 -1498.231} C_VEL
LIN {X 0,Y 587.341,Z 178.939,A -85,B 0,C 180,E1 -1500.868,E2 -1500.868} C_VEL
LIN {X 0,Y 587.306,Z 178.954,A -85,B 0,C 180,E1 -1503.721,E2 -1503.721} C_VEL
LIN {X 0,Y 587.37,Z 179.247,A -85,B 0,C 180,E1 -1504.054,E2 -1504.054} C_VEL
LIN {X 0,Y 588.391,Z 183.226,A -85,B 0,C 180,E1 -1504.533,E2 -1504.533} C_VEL
LIN {X 0,Y 588.234,Z 204.821,A -85,B 0,C 180,E1 -1506.78,E2 -1506.78} C_VEL
LIN {X 0,Y 588.014,Z 231.815,A -85,B 0,C 180,E1 -1509.538,E2 -1509.538} C_VEL
LIN {X 0,Y 587.922,Z 244.896,A -85,B 0,C 180,E1 -1510.84,E2 -1510.84} C_VEL
LIN {X 0,Y 588.611,Z 249.626,A -85,B 0,C 180,E1 -1510.943,E2 -1510.943} C_VEL
LIN {X 0,Y 588.306,Z 412.254,A -85,B 0,C 180,E1 -1512.997,E2 -1512.997} C_VEL
LIN {X 0,Y 588.223,Z 427.726,A -85,B 0,C 180,E1 -1513.337,E2 -1513.337} C_VEL
LIN {X 0,Y 588.082,Z 443.056,A -85,B 0,C 180,E1 -1513.824,E2 -1513.824} C_VEL
LIN {X 0,Y 587.975,Z 456.777,A -85,B 0,C 180,E1 -1514.399,E2 -1514.399} C_VEL
LIN {X 0,Y 587.839,Z 470.248,A -85,B 0,C 180,E1 -1515.106,E2 -1515.106} C_VEL
LIN {X 0,Y 587.739,Z 483.121,A -85,B 0,C 180,E1 -1515.93,E2 -1515.93} C_VEL
LIN {X 0,Y 587.582,Z 495.293,A -85,B 0,C 180,E1 -1516.865,E2 -1516.865} C_VEL
LIN {X 0,Y 587.453,Z 506.753,A -85,B 0,C 180,E1 -1517.916,E2 -1517.916} C_VEL
LIN {X 0,Y 587.348,Z 516.394,A -85,B 0,C 180,E1 -1518.963,E2 -1518.963} C_VEL
LIN {X 0,Y 587.305,Z 525.859,A -85,B 0,C 180,E1 -1520.182,E2 -1520.182} C_VEL
LIN {X 0,Y 587.265,Z 533.734,A -85,B 0,C 180,E1 -1521.397,E2 -1521.397} C_VEL
LIN {X 0,Y 587.215,Z 541.09,A -85,B 0,C 180,E1 -1522.781,E2 -1522.781} C_VEL
LIN {X 0,Y 587.227,Z 546.925,A -85,B 0,C 180,E1 -1524.162,E2 -1524.162} C_VEL
LIN {X 0,Y 587.136,Z 550.385,A -85,B 0,C 180,E1 -1525.194,E2 -1525.194} C_VEL
LIN {X 0,Y 587.179,Z 553.889,A -85,B 0,C 180,E1 -1526.569,E2 -1526.569} C_VEL
LIN {X 0,Y 587.14,Z 556.193,A -85,B 0,C 180,E1 -1527.942,E2 -1527.942} C_VEL
LIN {X 0,Y 587.137,Z 557.35,A -85,B 0,C 180,E1 -1529.314,E2 -1529.314} C_VEL
LIN {X 0,Y 587.137,Z 557.349,A -85,B 0,C 180,E1 -1530.686,E2 -1530.686} C_VEL
LIN {X 0,Y 587.14,Z 556.192,A -85,B 0,C 180,E1 -1532.058,E2 -1532.058} C_VEL
LIN {X 0,Y 587.179,Z 553.886,A -85,B 0,C 180,E1 -1533.431,E2 -1533.431} C_VEL
LIN {X 0,Y 587.136,Z 550.384,A -85,B 0,C 180,E1 -1534.807,E2 -1534.807} C_VEL
LIN {X 0,Y 587.18,Z 545.607,A -85,B 0,C 180,E1 -1536.184,E2 -1536.184} C_VEL
LIN {X 0,Y 587.23,Z 539.423,A -85,B 0,C 180,E1 -1537.565,E2 -1537.565} C_VEL
LIN {X 0,Y 587.266,Z 531.649,A -85,B 0,C 180,E1 -1538.95,E2 -1538.95} C_VEL
LIN {X 0,Y 587.351,Z 523.369,A -85,B 0,C 180,E1 -1540.166,E2 -1540.166} C_VEL
LIN {X 0,Y 587.4,Z 513.394,A -85,B 0,C 180,E1 -1541.386,E2 -1541.386} C_VEL
LIN {X 0,Y 587.522,Z 503.189,A -85,B 0,C 180,E1 -1542.434,E2 -1542.434} C_VEL
LIN {X 0,Y 587.629,Z 491.017,A -85,B 0,C 180,E1 -1543.487,E2 -1543.487} C_VEL
LIN {X 0,Y 587.774,Z 478.056,A -85,B 0,C 180,E1 -1544.416,E2 -1544.416} C_VEL
LIN {X 0,Y 587.912,Z 463.866,A -85,B 0,C 180,E1 -1545.248,E2 -1545.248} C_VEL
LIN {X 0,Y 588.033,Z 449.795,A -85,B 0,C 180,E1 -1545.911,E2 -1545.911} C_VEL
LIN {X 0,Y 588.169,Z 435.302,A -85,B 0,C 180,E1 -1546.442,E2 -1546.442} C_VEL
LIN {X 0,Y 588.271,Z 420.196,A -85,B 0,C 180,E1 -1546.847,E2 -1546.847} C_VEL
LIN {X 0,Y 588.326,Z 404.961,A -85,B 0,C 180,E1 -1547.111,E2 -1547.111} C_VEL
LIN {X 0,Y 588.56,Z 248.808,A -85,B 0,C 180,E1 -1549.069,E2 -1549.069} C_VEL
LIN {X 0,Y 587.924,Z 244.889,A -85,B 0,C 180,E1 -1549.161,E2 -1549.161} C_VEL
LIN {X 0,Y 588.143,Z 217.413,A -85,B 0,C 180,E1 -1551.927,E2 -1551.927} C_VEL
LIN {X 0,Y 588.418,Z 188.801,A -85,B 0,C 180,E1 -1554.88,E2 -1554.88} C_VEL
LIN {X 0,Y 588.392,Z 183.221,A -85,B 0,C 180,E1 -1555.467,E2 -1555.467} C_VEL
LIN {X 0,Y 587.336,Z 179.077,A -85,B 0,C 180,E1 -1555.986,E2 -1555.986} C_VEL
LIN {X 0,Y 587.307,Z 178.952,A -85,B 0,C 180,E1 -1558.598,E2 -1558.598} C_VEL
LIN {X 0,Y 587.319,Z 178.942,A -85,B 0,C 180,E1 -1560.967,E2 -1560.967} C_VEL
LIN {X 0,Y 587.324,Z 178.949,A -85,B 0,C 180,E1 -1563.397,E2 -1563.397} C_VEL
LIN {X 0,Y 587.286,Z 178.949,A -85,B 0,C 180,E1 -1565.9,E2 -1565.9} C_VEL
LIN {X 0,Y 587.316,Z 178.95,A -85,B 0,C 180,E1 -1568.48,E2 -1568.48} C_VEL
LIN {X 0,Y 587.333,Z 178.948,A -85,B 0,C 180,E1 -1571.157,E2 -1571.157} C_VEL
LIN {X 0,Y 587.309,Z 178.948,A -85,B 0,C 180,E1 -1574.112,E2 -1574.112} C_VEL
LIN {X 0,Y 587.309,Z 178.951,A -85,B 0,C 180,E1 -1576.993,E2 -1576.993} C_VEL
LIN {X 0,Y 587.31,Z 178.947,A -85,B 0,C 180,E1 -1579.745,E2 -1579.745} C_VEL
LIN {X 0,Y 587.339,Z 178.95,A -85,B 0,C 180,E1 -1582.392,E2 -1582.392} C_VEL
LIN {X 0,Y 587.349,Z 178.942,A -85,B 0,C 180,E1 -1585.652,E2 -1585.652} C_VEL
LIN {X 0,Y 587.344,Z 178.947,A -85,B 0,C 180,E1 -1588.231,E2 -1588.231} C_VEL
LIN {X 0,Y 587.344,Z 178.944,A -85,B 0,C 180,E1 -1590.867,E2 -1590.867} C_VEL
LIN {X 0,Y 587.358,Z 178.941,A -85,B 0,C 180,E1 -1593.818,E2 -1593.818} C_VEL
LIN {X 0,Y 587.331,Z 178.95,A -85,B 0,C 180,E1 -1595.993,E2 -1595.993} C_VEL
LIN {X 0,Y 587.312,Z 178.955,A -85,B 0,C 180,E1 -1598.225,E2 -1598.225} C_VEL
LIN {X 0,Y 587.341,Z 178.943,A -85,B 0,C 180,E1 -1601.151,E2 -1601.151} C_VEL
LIN {X 0,Y 587.323,Z 178.945,A -85,B 0,C 180,E1 -1603.31,E2 -1603.31} C_VEL
LIN {X 0,Y 587.359,Z 178.947,A -85,B 0,C 180,E1 -1606.154,E2 -1606.154} C_VEL
LIN {X 0,Y 587.332,Z 178.944,A -85,B 0,C 180,E1 -1608.962,E2 -1608.962} C_VEL
LIN {X 0,Y 587.362,Z 178.948,A -85,B 0,C 180,E1 -1611.745,E2 -1611.745} C_VEL
LIN {X 0,Y 587.356,Z 178.941,A -85,B 0,C 180,E1 -1614.507,E2 -1614.507} C_VEL
LIN {X 0,Y 587.365,Z 178.943,A -85,B 0,C 180,E1 -1617.257,E2 -1617.257} C_VEL
LIN {X 0,Y 587.38,Z 178.942,A -85,B 0,C 180,E1 -1620,E2 -1620} C_VEL
LIN {X 0,Y 587.373,Z 178.938,A -85,B 0,C 180,E1 -1622.743,E2 -1622.743} C_VEL
LIN {X 0,Y 587.353,Z 178.951,A -85,B 0,C 180,E1 -1625.493,E2 -1625.493} C_VEL
LIN {X 0,Y 587.367,Z 178.939,A -85,B 0,C 180,E1 -1628.255,E2 -1628.255} C_VEL
LIN {X 0,Y 587.345,Z 178.948,A -85,B 0,C 180,E1 -1631.134,E2 -1631.134} C_VEL
LIN {X 0,Y 587.362,Z 178.94,A -85,B 0,C 180,E1 -1634.261,E2 -1634.261} C_VEL
LIN {X 0,Y 587.349,Z 178.949,A -85,B 0,C 180,E1 -1637.406,E2 -1637.406} C_VEL
LIN {X 0,Y 587.307,Z 178.947,A -85,B 0,C 180,E1 -1638.315,E2 -1638.315} C_VEL
LIN {X 0,Y 586.664,Z 179.033,A -85,B 0,C 180,E1 -1638.887,E2 -1638.887} C_VEL
LIN {X 0,Y 583.838,Z 179.391,A -85,B 0,C 180,E1 -1639.815,E2 -1639.815} C_VEL
LIN {X 0,Y 581.428,Z 179.693,A -85,B 0,C 180,E1 -1640.562,E2 -1640.562} C_VEL
LIN {X 0,Y 580.375,Z 179.82,A -85,B 0,C 180,E1 -1641.139,E2 -1641.139} C_VEL
LIN {X 0,Y 580.28,Z 179.829,A -85,B 0,C 180,E1 -1641.334,E2 -1641.334} C_VEL
LIN {X 0,Y 580.299,Z 179.82,A -85,B 0,C 180,E1 -1644.316,E2 -1644.316} C_VEL
LIN {X 0,Y 580.275,Z 179.827,A -85,B 0,C 180,E1 -1646.624,E2 -1646.624} C_VEL
LIN {X 0,Y 580.3,Z 179.822,A -85,B 0,C 180,E1 -1649.31,E2 -1649.31} C_VEL
LIN {X 0,Y 580.295,Z 179.822,A -85,B 0,C 180,E1 -1652.201,E2 -1652.201} C_VEL
LIN {X 0,Y 580.301,Z 179.827,A -85,B 0,C 180,E1 -1654.696,E2 -1654.696} C_VEL
LIN {X 0,Y 580.298,Z 179.822,A -85,B 0,C 180,E1 -1657.269,E2 -1657.269} C_VEL
LIN {X 0,Y 580.291,Z 179.823,A -85,B 0,C 180,E1 -1660.271,E2 -1660.271} C_VEL
LIN {X 0,Y 580.276,Z 179.831,A -85,B 0,C 180,E1 -1662.707,E2 -1662.707} C_VEL
LIN {X 0,Y 580.267,Z 179.824,A -85,B 0,C 180,E1 -1665.61,E2 -1665.61} C_VEL
LIN {X 0,Y 580.314,Z 179.823,A -85,B 0,C 180,E1 -1668.235,E2 -1668.235} C_VEL
LIN {X 0,Y 580.272,Z 179.825,A -85,B 0,C 180,E1 -1670.965,E2 -1670.965} C_VEL
LIN {X 0,Y 580.271,Z 179.824,A -85,B 0,C 180,E1 -1673.597,E2 -1673.597} C_VEL
LIN {X 0,Y 580.315,Z 179.826,A -85,B 0,C 180,E1 -1676.145,E2 -1676.145} C_VEL
LIN {X 0,Y 580.276,Z 179.827,A -85,B 0,C 180,E1 -1678.615,E2 -1678.615} C_VEL
LIN {X 0,Y 580.291,Z 179.823,A -85,B 0,C 180,E1 -1681.024,E2 -1681.024} C_VEL
LIN {X 0,Y 580.279,Z 179.83,A -85,B 0,C 180,E1 -1684.15,E2 -1684.15} C_VEL
LIN {X 0,Y 580.316,Z 180.046,A -85,B 0,C 180,E1 -1685.188,E2 -1685.188} C_VEL
LIN {X 0,Y 581.252,Z 185.059,A -85,B 0,C 180,E1 -1685.916,E2 -1685.916} C_VEL
LIN {X 0,Y 581,Z 206.684,A -85,B 0,C 180,E1 -1688.722,E2 -1688.722} C_VEL
LIN {X 0,Y 580.75,Z 229.849,A -85,B 0,C 180,E1 -1691.661,E2 -1691.661} C_VEL
LIN {X 0,Y 580.676,Z 244.606,A -85,B 0,C 180,E1 -1693.476,E2 -1693.476} C_VEL
LIN {X 0,Y 581.417,Z 250.411,A -85,B 0,C 180,E1 -1693.588,E2 -1693.588} C_VEL
LIN {X 0,Y 581.142,Z 382.872,A -85,B 0,C 180,E1 -1695.265,E2 -1695.265} C_VEL
LIN {X 0,Y 581.051,Z 397.13,A -85,B 0,C 180,E1 -1695.592,E2 -1695.592} C_VEL
LIN {X 0,Y 580.938,Z 410.7,A -85,B 0,C 180,E1 -1696.043,E2 -1696.043} C_VEL
LIN {X 0,Y 580.804,Z 423.752,A -85,B 0,C 180,E1 -1696.619,E2 -1696.619} C_VEL
LIN {X 0,Y 580.66,Z 436.387,A -85,B 0,C 180,E1 -1697.328,E2 -1697.328} C_VEL
LIN {X 0,Y 580.542,Z 447.89,A -85,B 0,C 180,E1 -1698.124,E2 -1698.124} C_VEL
LIN {X 0,Y 580.463,Z 458.452,A -85,B 0,C 180,E1 -1699.008,E2 -1699.008} C_VEL
LIN {X 0,Y 580.319,Z 468.917,A -85,B 0,C 180,E1 -1700.062,E2 -1700.062} C_VEL
LIN {X 0,Y 580.254,Z 477.565,A -85,B 0,C 180,E1 -1701.116,E2 -1701.116} C_VEL
LIN {X 0,Y 580.177,Z 485.852,A -85,B 0,C 180,E1 -1702.342,E2 -1702.342} C_VEL
LIN {X 0,Y 580.124,Z 491.757,A -85,B 0,C 180,E1 -1703.415,E2 -1703.415} C_VEL
LIN {X 0,Y 580.129,Z 496.383,A -85,B 0,C 180,E1 -1704.438,E2 -1704.438} C_VEL
LIN {X 0,Y 580.104,Z 501.307,A -85,B 0,C 180,E1 -1705.831,E2 -1705.831} C_VEL
LIN {X 0,Y 580.041,Z 504.741,A -85,B 0,C 180,E1 -1707.222,E2 -1707.222} C_VEL
LIN {X 0,Y 580.045,Z 506.783,A -85,B 0,C 180,E1 -1708.611,E2 -1708.611} C_VEL
LIN {X 0,Y 580.037,Z 507.496,A -85,B 0,C 180,E1 -1710,E2 -1710} C_VEL
LIN {X 0,Y 580.042,Z 506.882,A -85,B 0,C 180,E1 -1711.388,E2 -1711.388} C_VEL
LIN {X 0,Y 580.039,Z 504.927,A -85,B 0,C 180,E1 -1712.778,E2 -1712.778} C_VEL
LIN {X 0,Y 580.104,Z 501.582,A -85,B 0,C 180,E1 -1714.168,E2 -1714.168} C_VEL
LIN {X 0,Y 580.129,Z 496.753,A -85,B 0,C 180,E1 -1715.561,E2 -1715.561} C_VEL
LIN {X 0,Y 580.141,Z 490.288,A -85,B 0,C 180,E1 -1716.958,E2 -1716.958} C_VEL
LIN {X 0,Y 580.192,Z 483.089,A -85,B 0,C 180,E1 -1718.182,E2 -1718.182} C_VEL
LIN {X 0,Y 580.284,Z 475.55,A -85,B 0,C 180,E1 -1719.234,E2 -1719.234} C_VEL
LIN {X 0,Y 580.347,Z 466.5,A -85,B 0,C 180,E1 -1720.289,E2 -1720.289} C_VEL
LIN {X 0,Y 580.494,Z 455.541,A -85,B 0,C 180,E1 -1721.345,E2 -1721.345} C_VEL
LIN {X 0,Y 580.575,Z 444.369,A -85,B 0,C 180,E1 -1722.23,E2 -1722.23} C_VEL
LIN {X 0,Y 580.706,Z 432.023,A -85,B 0,C 180,E1 -1723.026,E2 -1723.026} C_VEL
LIN {X 0,Y 580.873,Z 420.145,A -85,B 0,C 180,E1 -1723.646,E2 -1723.646} C_VEL
LIN {X 0,Y 581.006,Z 407.165,A -85,B 0,C 180,E1 -1724.179,E2 -1724.179} C_VEL
LIN {X 0,Y 581.068,Z 392.999,A -85,B 0,C 180,E1 -1724.608,E2 -1724.608} C_VEL
LIN {X 0,Y 581.127,Z 378.673,A -85,B 0,C 180,E1 -1724.891,E2 -1724.891} C_VEL
LIN {X 0,Y 581.378,Z 249.337,A -85,B 0,C 180,E1 -1726.517,E2 -1726.517} C_VEL
LIN {X 0,Y 580.681,Z 244.608,A -85,B 0,C 180,E1 -1726.614,E2 -1726.614} C_VEL
LIN {X 0,Y 580.753,Z 227.67,A -85,B 0,C 180,E1 -1728.704,E2 -1728.704} C_VEL
LIN {X 0,Y 581.013,Z 206.087,A -85,B 0,C 180,E1 -1731.444,E2 -1731.444} C_VEL
LIN {X 0,Y 581.242,Z 185.747,A -85,B 0,C 180,E1 -1734.084,E2 -1734.084} C_VEL
LIN {X 0,Y 580.697,Z 181.734,A -85,B 0,C 180,E1 -1734.638,E2 -1734.638} C_VEL
LIN {X 0,Y 580.29,Z 179.982,A -85,B 0,C 180,E1 -1734.921,E2 -1734.921} C_VEL
LIN {X 0,Y 580.253,Z 179.828,A -85,B 0,C 180,E1 -1737.403,E2 -1737.403} C_VEL
LIN {X 0,Y 580.284,Z 179.828,A -85,B 0,C 180,E1 -1739.772,E2 -1739.772} C_VEL
LIN {X 0,Y 580.297,Z 179.823,A -85,B 0,C 180,E1 -1742.2,E2 -1742.2} C_VEL
LIN {X 0,Y 580.286,Z 179.822,A -85,B 0,C 180,E1 -1744.696,E2 -1744.696} C_VEL
LIN {X 0,Y 580.296,Z 179.823,A -85,B 0,C 180,E1 -1747.268,E2 -1747.268} C_VEL
LIN {X 0,Y 580.288,Z 179.823,A -85,B 0,C 180,E1 -1750.27,E2 -1750.27} C_VEL
LIN {X 0,Y 580.274,Z 179.822,A -85,B 0,C 180,E1 -1752.706,E2 -1752.706} C_VEL
LIN {X 0,Y 580.266,Z 179.832,A -85,B 0,C 180,E1 -1755.608,E2 -1755.608} C_VEL
LIN {X 0,Y 580.31,Z 179.819,A -85,B 0,C 180,E1 -1758.234,E2 -1758.234} C_VEL
LIN {X 0,Y 580.274,Z 179.825,A -85,B 0,C 180,E1 -1760.965,E2 -1760.965} C_VEL
LIN {X 0,Y 580.292,Z 179.826,A -85,B 0,C 180,E1 -1763.598,E2 -1763.598} C_VEL
LIN {X 0,Y 580.315,Z 179.817,A -85,B 0,C 180,E1 -1766.145,E2 -1766.145} C_VEL
LIN {X 0,Y 580.278,Z 179.825,A -85,B 0,C 180,E1 -1768.614,E2 -1768.614} C_VEL
LIN {X 0,Y 580.289,Z 179.828,A -85,B 0,C 180,E1 -1771.024,E2 -1771.024} C_VEL
LIN {X 0,Y 580.285,Z 179.823,A -85,B 0,C 180,E1 -1773.665,E2 -1773.665} C_VEL
LIN {X 0,Y 580.295,Z 179.821,A -85,B 0,C 180,E1 -1775.683,E2 -1775.683} C_VEL
LIN {X 0,Y 580.267,Z 179.824,A -85,B 0,C 180,E1 -1777.947,E2 -1777.947} C_VEL
LIN {X 0,Y 580.312,Z 179.828,A -85,B 0,C 180,E1 -1780.914,E2 -1780.914} C_VEL
LIN {X 0,Y 580.276,Z 179.822,A -85,B 0,C 180,E1 -1783.825,E2 -1783.825} C_VEL
LIN {X 0,Y 580.321,Z 179.818,A -85,B 0,C 180,E1 -1785.983,E2 -1785.983} C_VEL
LIN {X 0,Y 580.296,Z 179.828,A -85,B 0,C 180,E1 -1788.827,E2 -1788.827} C_VEL
LIN {X 0,Y 580.328,Z 179.816,A -85,B 0,C 180,E1 -1791.644,E2 -1791.644} C_VEL
LIN {X 0,Y 580.319,Z 179.825,A -85,B 0,C 180,E1 -1794.44,E2 -1794.44} C_VEL
LIN {X 0,Y 580.338,Z 179.815,A -85,B 0,C 180,E1 -1797.223,E2 -1797.223} C_VEL
LIN {X 0,Y 580.345,Z 179.818,A -85,B 0,C 180,E1 -1800,E2 -1800} C_VEL
LIN {X 0,Y 580.334,Z 179.819,A -85,B 0,C 180,E1 -1802.776,E2 -1802.776} C_VEL
LIN {X 0,Y 580.321,Z 179.817,A -85,B 0,C 180,E1 -1805.56,E2 -1805.56} C_VEL
LIN {X 0,Y 580.327,Z 179.823,A -85,B 0,C 180,E1 -1808.356,E2 -1808.356} C_VEL
LIN {X 0,Y 580.291,Z 179.821,A -85,B 0,C 180,E1 -1811.191,E2 -1811.191} C_VEL
LIN {X 0,Y 580.32,Z 179.826,A -85,B 0,C 180,E1 -1814.017,E2 -1814.017} C_VEL
LIN {X 0,Y 580.304,Z 179.819,A -85,B 0,C 180,E1 -1816.914,E2 -1816.914} C_VEL
LIN {X 0,Y 580.297,Z 179.829,A -85,B 0,C 180,E1 -1819.822,E2 -1819.822} C_VEL
LIN {X 0,Y 580.288,Z 179.821,A -85,B 0,C 180,E1 -1822.803,E2 -1822.803} C_VEL
LIN {X 0,Y 580.302,Z 179.82,A -85,B 0,C 180,E1 -1825.08,E2 -1825.08} C_VEL
LIN {X 0,Y 580.291,Z 179.829,A -85,B 0,C 180,E1 -1827.859,E2 -1827.859} C_VEL
LIN {X 0,Y 580.278,Z 179.822,A -85,B 0,C 180,E1 -1830.695,E2 -1830.695} C_VEL
LIN {X 0,Y 580.297,Z 179.823,A -85,B 0,C 180,E1 -1833.317,E2 -1833.317} C_VEL
LIN {X 0,Y 580.264,Z 179.83,A -85,B 0,C 180,E1 -1835.76,E2 -1835.76} C_VEL
LIN {X 0,Y 580.28,Z 179.823,A -85,B 0,C 180,E1 -1838.147,E2 -1838.147} C_VEL
LIN {X 0,Y 580.293,Z 179.823,A -85,B 0,C 180,E1 -1840.844,E2 -1840.844} C_VEL
LIN {X 0,Y 580.266,Z 179.829,A -85,B 0,C 180,E1 -1843.659,E2 -1843.659} C_VEL
LIN {X 0,Y 580.268,Z 179.825,A -85,B 0,C 180,E1 -1846.61,E2 -1846.61} C_VEL
LIN {X 0,Y 580.292,Z 179.827,A -85,B 0,C 180,E1 -1849.157,E2 -1849.157} C_VEL
LIN {X 0,Y 580.28,Z 179.823,A -85,B 0,C 180,E1 -1851.928,E2 -1851.928} C_VEL
LIN {X 0,Y 580.246,Z 179.827,A -85,B 0,C 180,E1 -1854.453,E2 -1854.453} C_VEL
LIN {X 0,Y 580.282,Z 179.832,A -85,B 0,C 180,E1 -1856.975,E2 -1856.975} C_VEL
LIN {X 0,Y 580.277,Z 179.811,A -85,B 0,C 180,E1 -1859.425,E2 -1859.425} C_VEL
LIN {X 0,Y 580.284,Z 179.826,A -85,B 0,C 180,E1 -1862.144,E2 -1862.144} C_VEL
LIN {X 0,Y 580.312,Z 180.014,A -85,B 0,C 180,E1 -1863.8,E2 -1863.8} C_VEL
LIN {X 0,Y 581.575,Z 184.957,A -85,B 0,C 180,E1 -1864.405,E2 -1864.405} C_VEL
LIN {X 0,Y 581.472,Z 203.022,A -85,B 0,C 180,E1 -1866.305,E2 -1866.305} C_VEL
LIN {X 0,Y 581.171,Z 230.015,A -85,B 0,C 180,E1 -1869.101,E2 -1869.101} C_VEL
LIN {X 0,Y 581.056,Z 244.931,A -85,B 0,C 180,E1 -1870.606,E2 -1870.606} C_VEL
LIN {X 0,Y 581.9,Z 250.832,A -85,B 0,C 180,E1 -1870.73,E2 -1870.73} C_VEL
LIN {X 0,Y 581.538,Z 412.327,A -85,B 0,C 180,E1 -1872.795,E2 -1872.795} C_VEL
LIN {X 0,Y 581.432,Z 427.724,A -85,B 0,C 180,E1 -1873.137,E2 -1873.137} C_VEL
LIN {X 0,Y 581.255,Z 443.054,A -85,B 0,C 180,E1 -1873.628,E2 -1873.628} C_VEL
LIN {X 0,Y 581.121,Z 456.78,A -85,B 0,C 180,E1 -1874.211,E2 -1874.211} C_VEL
LIN {X 0,Y 580.949,Z 470.251,A -85,B 0,C 180,E1 -1874.925,E2 -1874.925} C_VEL
LIN {X 0,Y 580.803,Z 483.487,A -85,B 0,C 180,E1 -1875.784,E2 -1875.784} C_VEL
LIN {X 0,Y 580.608,Z 495.294,A -85,B 0,C 180,E1 -1876.704,E2 -1876.704} C_VEL
LIN {X 0,Y 580.478,Z 506.753,A -85,B 0,C 180,E1 -1877.768,E2 -1877.768} C_VEL
LIN {X 0,Y 580.307,Z 517.453,A -85,B 0,C 180,E1 -1878.953,E2 -1878.953} C_VEL
LIN {X 0,Y 580.268,Z 525.86,A -85,B 0,C 180,E1 -1880.062,E2 -1880.062} C_VEL
LIN {X 0,Y 580.214,Z 533.735,A -85,B 0,C 180,E1 -1881.292,E2 -1881.292} C_VEL
LIN {X 0,Y 580.13,Z 541.091,A -85,B 0,C 180,E1 -1882.692,E2 -1882.692} C_VEL
LIN {X 0,Y 580.132,Z 546.924,A -85,B 0,C 180,E1 -1884.09,E2 -1884.09} C_VEL
LIN {X 0,Y 580.041,Z 550.386,A -85,B 0,C 180,E1 -1885.135,E2 -1885.135} C_VEL
LIN {X 0,Y 580.104,Z 553.889,A -85,B 0,C 180,E1 -1886.527,E2 -1886.527} C_VEL
LIN {X 0,Y 580.039,Z 556.193,A -85,B 0,C 180,E1 -1887.917,E2 -1887.917} C_VEL
LIN {X 0,Y 580.038,Z 557.349,A -85,B 0,C 180,E1 -1889.306,E2 -1889.306} C_VEL
LIN {X 0,Y 580.038,Z 557.349,A -85,B 0,C 180,E1 -1890.694,E2 -1890.694} C_VEL
LIN {X 0,Y 580.039,Z 556.191,A -85,B 0,C 180,E1 -1892.083,E2 -1892.083} C_VEL
LIN {X 0,Y 580.104,Z 553.886,A -85,B 0,C 180,E1 -1893.473,E2 -1893.473} C_VEL
LIN {X 0,Y 580.041,Z 550.384,A -85,B 0,C 180,E1 -1894.866,E2 -1894.866} C_VEL
LIN {X 0,Y 580.093,Z 545.608,A -85,B 0,C 180,E1 -1896.26,E2 -1896.26} C_VEL
LIN {X 0,Y 580.165,Z 539.422,A -85,B 0,C 180,E1 -1897.658,E2 -1897.658} C_VEL
LIN {X 0,Y 580.207,Z 531.648,A -85,B 0,C 180,E1 -1899.06,E2 -1899.06} C_VEL
LIN {X 0,Y 580.309,Z 523.368,A -85,B 0,C 180,E1 -1900.29,E2 -1900.29} C_VEL
LIN {X 0,Y 580.383,Z 513.394,A -85,B 0,C 180,E1 -1901.525,E2 -1901.525} C_VEL
LIN {X 0,Y 580.541,Z 503.188,A -85,B 0,C 180,E1 -1902.586,E2 -1902.586} C_VEL
LIN {X 0,Y 580.678,Z 491.018,A -85,B 0,C 180,E1 -1903.651,E2 -1903.651} C_VEL
LIN {X 0,Y 580.875,Z 477.527,A -85,B 0,C 180,E1 -1904.625,E2 -1904.625} C_VEL
LIN {X 0,Y 581.029,Z 463.868,A -85,B 0,C 180,E1 -1905.433,E2 -1905.433} C_VEL
LIN {X 0,Y 581.185,Z 449.797,A -85,B 0,C 180,E1 -1906.103,E2 -1906.103} C_VEL
LIN {X 0,Y 581.368,Z 435.303,A -85,B 0,C 180,E1 -1906.64,E2 -1906.64} C_VEL
LIN {X 0,Y 581.499,Z 419.971,A -85,B 0,C 180,E1 -1907.054,E2 -1907.054} C_VEL
LIN {X 0,Y 581.558,Z 404.428,A -85,B 0,C 180,E1 -1907.325,E2 -1907.325} C_VEL
LIN {X 0,Y 581.883,Z 249.725,A -85,B 0,C 180,E1 -1909.285,E2 -1909.285} C_VEL
LIN {X 0,Y 581.046,Z 244.786,A -85,B 0,C 180,E1 -1909.405,E2 -1909.405} C_VEL
LIN {X 0,Y 581.329,Z 217.413,A -85,B 0,C 180,E1 -1912.197,E2 -1912.197} C_VEL
LIN {X 0,Y 581.698,Z 188.578,A -85,B 0,C 180,E1 -1915.207,E2 -1915.207} C_VEL
LIN {X 0,Y 581.576,Z 184.951,A -85,B 0,C 180,E1 -1915.596,E2 -1915.596} C_VEL
LIN {X 0,Y 580.284,Z 179.961,A -85,B 0,C 180,E1 -1916.215,E2 -1916.215} C_VEL
LIN {X 0,Y 580.282,Z 179.814,A -85,B 0,C 180,E1 -1918.977,E2 -1918.977} C_VEL
LIN {X 0,Y 580.297,Z 179.819,A -85,B 0,C 180,E1 -1922.03,E2 -1922.03} C_VEL
LIN {X 0,Y 580.284,Z 179.828,A -85,B 0,C 180,E1 -1924.696,E2 -1924.696} C_VEL
LIN {X 0,Y 580.294,Z 179.825,A -85,B 0,C 180,E1 -1927.268,E2 -1927.268} C_VEL
LIN {X 0,Y 580.285,Z 179.818,A -85,B 0,C 180,E1 -1930.27,E2 -1930.27} C_VEL
LIN {X 0,Y 580.274,Z 179.832,A -85,B 0,C 180,E1 -1932.706,E2 -1932.706} C_VEL
LIN {X 0,Y 580.252,Z 179.826,A -85,B 0,C 180,E1 -1935.61,E2 -1935.61} C_VEL
LIN {X 0,Y 580.274,Z 179.826,A -85,B 0,C 180,E1 -1938.231,E2 -1938.231} C_VEL
LIN {X 0,Y 580.28,Z 179.826,A -85,B 0,C 180,E1 -1940.965,E2 -1940.965} C_VEL
LIN {X 0,Y 580.265,Z 179.824,A -85,B 0,C 180,E1 -1943.596,E2 -1943.596} C_VEL
LIN {X 0,Y 580.304,Z 179.825,A -85,B 0,C 180,E1 -1946.145,E2 -1946.145} C_VEL
LIN {X 0,Y 580.279,Z 179.829,A -85,B 0,C 180,E1 -1948.615,E2 -1948.615} C_VEL
LIN {X 0,Y 580.287,Z 179.822,A -85,B 0,C 180,E1 -1951.024,E2 -1951.024} C_VEL
LIN {X 0,Y 580.29,Z 179.819,A -85,B 0,C 180,E1 -1953.666,E2 -1953.666} C_VEL
LIN {X 0,Y 580.296,Z 179.822,A -85,B 0,C 180,E1 -1955.684,E2 -1955.684} C_VEL
LIN {X 0,Y 580.264,Z 179.831,A -85,B 0,C 180,E1 -1957.947,E2 -1957.947} C_VEL
LIN {X 0,Y 580.294,Z 179.821,A -85,B 0,C 180,E1 -1960.913,E2 -1960.913} C_VEL
LIN {X 0,Y 580.3,Z 179.819,A -85,B 0,C 180,E1 -1963.102,E2 -1963.102} C_VEL
LIN {X 0,Y 580.324,Z 179.826,A -85,B 0,C 180,E1 -1965.983,E2 -1965.983} C_VEL
LIN {X 0,Y 580.301,Z 179.82,A -85,B 0,C 180,E1 -1968.827,E2 -1968.827} C_VEL
LIN {X 0,Y 580.324,Z 179.823,A -85,B 0,C 180,E1 -1971.644,E2 -1971.644} C_VEL
LIN {X 0,Y 580.321,Z 179.817,A -85,B 0,C 180,E1 -1974.44,E2 -1974.44} C_VEL
LIN {X 0,Y 580.332,Z 179.819,A -85,B 0,C 180,E1 -1977.224,E2 -1977.224} C_VEL
LIN {X 0,Y 580.35,Z 179.818,A -85,B 0,C 180,E1 -1980,E2 -1980} C_VEL
LIN {X 0,Y 580.339,Z 179.815,A -85,B 0,C 180,E1 -1982.777,E2 -1982.777} C_VEL
LIN {X 0,Y 580.32,Z 179.826,A -85,B 0,C 180,E1 -1985.56,E2 -1985.56} C_VEL
LIN {X 0,Y 580.33,Z 179.816,A -85,B 0,C 180,E1 -1988.356,E2 -1988.356} C_VEL
LIN {X 0,Y 580.297,Z 179.827,A -85,B 0,C 180,E1 -1991.191,E2 -1991.191} C_VEL
LIN {X 0,Y 580.324,Z 179.818,A -85,B 0,C 180,E1 -1994.017,E2 -1994.017} C_VEL
LIN {X 0,Y 580.309,Z 179.823,A -85,B 0,C 180,E1 -1996.914,E2 -1996.914} C_VEL
LIN {X 0,Y 580.303,Z 179.82,A -85,B 0,C 180,E1 -1999.823,E2 -1999.823} C_VEL
LIN {X 0,Y 580.28,Z 179.829,A -85,B 0,C 180,E1 -2001.334,E2 -2001.334} C_VEL
LIN {X 0,Y 579.584,Z 179.912,A -85,B 0,C 180,E1 -2001.913,E2 -2001.913} C_VEL
LIN {X 0,Y 576.708,Z 180.274,A -85,B 0,C 180,E1 -2002.853,E2 -2002.853} C_VEL
LIN {X 0,Y 574.314,Z 180.567,A -85,B 0,C 180,E1 -2003.609,E2 -2003.609} C_VEL
LIN {X 0,Y 573.315,Z 180.69,A -85,B 0,C 180,E1 -2004.193,E2 -2004.193} C_VEL
LIN {X 0,Y 573.248,Z 180.699,A -85,B 0,C 180,E1 -2004.391,E2 -2004.391} C_VEL
LIN {X 0,Y 573.249,Z 180.706,A -85,B 0,C 180,E1 -2006.976,E2 -2006.976} C_VEL
LIN {X 0,Y 573.245,Z 180.699,A -85,B 0,C 180,E1 -2009.489,E2 -2009.489} C_VEL
LIN {X 0,Y 573.251,Z 180.705,A -85,B 0,C 180,E1 -2012.645,E2 -2012.645} C_VEL
LIN {X 0,Y 573.268,Z 180.698,A -85,B 0,C 180,E1 -2015.184,E2 -2015.184} C_VEL
LIN {X 0,Y 573.235,Z 180.7,A -85,B 0,C 180,E1 -2017.808,E2 -2017.808} C_VEL
LIN {X 0,Y 573.244,Z 180.704,A -85,B 0,C 180,E1 -2020.525,E2 -2020.525} C_VEL
LIN {X 0,Y 573.235,Z 180.7,A -85,B 0,C 180,E1 -2023.36,E2 -2023.36} C_VEL
LIN {X 0,Y 573.244,Z 180.706,A -85,B 0,C 180,E1 -2026.331,E2 -2026.331} C_VEL
LIN {X 0,Y 573.244,Z 180.708,A -85,B 0,C 180,E1 -2028.545,E2 -2028.545} C_VEL
LIN {X 0,Y 573.238,Z 180.7,A -85,B 0,C 180,E1 -2031.298,E2 -2031.298} C_VEL
LIN {X 0,Y 573.239,Z 180.704,A -85,B 0,C 180,E1 -2034.015,E2 -2034.015} C_VEL
LIN {X 0,Y 573.271,Z 180.698,A -85,B 0,C 180,E1 -2036.518,E2 -2036.518} C_VEL
LIN {X 0,Y 573.228,Z 180.702,A -85,B 0,C 180,E1 -2039.118,E2 -2039.118} C_VEL
LIN {X 0,Y 573.228,Z 180.704,A -85,B 0,C 180,E1 -2041.435,E2 -2041.435} C_VEL
LIN {X 0,Y 573.242,Z 180.703,A -85,B 0,C 180,E1 -2044.589,E2 -2044.589} C_VEL
LIN {X 0,Y 573.293,Z 180.931,A -85,B 0,C 180,E1 -2044.973,E2 -2044.973} C_VEL
LIN {X 0,Y 574.424,Z 186.6,A -85,B 0,C 180,E1 -2045.804,E2 -2045.804} C_VEL
LIN {X 0,Y 574.113,Z 207.966,A -85,B 0,C 180,E1 -2048.616,E2 -2048.616} C_VEL
LIN {X 0,Y 573.792,Z 231.301,A -85,B 0,C 180,E1 -2051.615,E2 -2051.615} C_VEL
LIN {X 0,Y 573.697,Z 244.299,A -85,B 0,C 180,E1 -2053.246,E2 -2053.246} C_VEL
LIN {X 0,Y 574.285,Z 248.024,A -85,B 0,C 180,E1 -2053.347,E2 -2053.347} C_VEL
LIN {X 0,Y 574.579,Z 252.245,A -85,B 0,C 180,E1 -2053.409,E2 -2053.409} C_VEL
LIN {X 0,Y 574.281,Z 382.901,A -85,B 0,C 180,E1 -2055.085,E2 -2055.085} C_VEL
LIN {X 0,Y 574.174,Z 397.306,A -85,B 0,C 180,E1 -2055.42,E2 -2055.42} C_VEL
LIN {X 0,Y 574.031,Z 411.841,A -85,B 0,C 180,E1 -2055.917,E2 -2055.917} C_VEL
LIN {X 0,Y 573.848,Z 425.522,A -85,B 0,C 180,E1 -2056.544,E2 -2056.544} C_VEL
LIN {X 0,Y 573.687,Z 437.81,A -85,B 0,C 180,E1 -2057.261,E2 -2057.261} C_VEL
LIN {X 0,Y 573.551,Z 450.211,A -85,B 0,C 180,E1 -2058.156,E2 -2058.156} C_VEL
LIN {X 0,Y 573.438,Z 460.705,A -85,B 0,C 180,E1 -2059.081,E2 -2059.081} C_VEL
LIN {X 0,Y 573.245,Z 470.475,A -85,B 0,C 180,E1 -2060.117,E2 -2060.117} C_VEL
LIN {X 0,Y 573.202,Z 478.858,A -85,B 0,C 180,E1 -2061.184,E2 -2061.184} C_VEL
LIN {X 0,Y 573.111,Z 486.87,A -85,B 0,C 180,E1 -2062.425,E2 -2062.425} C_VEL
LIN {X 0,Y 573.022,Z 493.322,A -85,B 0,C 180,E1 -2063.662,E2 -2063.662} C_VEL
LIN {X 0,Y 573,Z 497.797,A -85,B 0,C 180,E1 -2064.722,E2 -2064.722} C_VEL
LIN {X 0,Y 573.029,Z 501.31,A -85,B 0,C 180,E1 -2065.78,E2 -2065.78} C_VEL
LIN {X 0,Y 572.957,Z 504.743,A -85,B 0,C 180,E1 -2067.187,E2 -2067.187} C_VEL
LIN {X 0,Y 572.944,Z 506.785,A -85,B 0,C 180,E1 -2068.594,E2 -2068.594} C_VEL
LIN {X 0,Y 572.937,Z 507.496,A -85,B 0,C 180,E1 -2070,E2 -2070} C_VEL
LIN {X 0,Y 572.942,Z 506.882,A -85,B 0,C 180,E1 -2071.406,E2 -2071.406} C_VEL
LIN {X 0,Y 572.954,Z 504.927,A -85,B 0,C 180,E1 -2072.812,E2 -2072.812} C_VEL
LIN {X 0,Y 573.03,Z 501.581,A -85,B 0,C 180,E1 -2074.22,E2 -2074.22} C_VEL
LIN {X 0,Y 573.056,Z 496.75,A -85,B 0,C 180,E1 -2075.63,E2 -2075.63} C_VEL
LIN {X 0,Y 573.054,Z 490.286,A -85,B 0,C 180,E1 -2077.044,E2 -2077.044} C_VEL
LIN {X 0,Y 573.142,Z 483.086,A -85,B 0,C 180,E1 -2078.284,E2 -2078.284} C_VEL
LIN {X 0,Y 573.225,Z 474.186,A -85,B 0,C 180,E1 -2079.527,E2 -2079.527} C_VEL
LIN {X 0,Y 573.35,Z 464.845,A -85,B 0,C 180,E1 -2080.595,E2 -2080.595} C_VEL
LIN {X 0,Y 573.476,Z 454.497,A -85,B 0,C 180,E1 -2081.576,E2 -2081.576} C_VEL
LIN {X 0,Y 573.626,Z 443.087,A -85,B 0,C 180,E1 -2082.47,E2 -2082.47} C_VEL
LIN {X 0,Y 573.802,Z 430.444,A -85,B 0,C 180,E1 -2083.276,E2 -2083.276} C_VEL
LIN {X 0,Y 573.99,Z 418.159,A -85,B 0,C 180,E1 -2083.903,E2 -2083.903} C_VEL
LIN {X 0,Y 574.151,Z 404.334,A -85,B 0,C 180,E1 -2084.45,E2 -2084.45} C_VEL
LIN {X 0,Y 574.242,Z 390.375,A -85,B 0,C 180,E1 -2084.849,E2 -2084.849} C_VEL
LIN {X 0,Y 574.298,Z 375.609,A -85,B 0,C 180,E1 -2085.118,E2 -2085.118} C_VEL
LIN {X 0,Y 574.502,Z 249.292,A -85,B 0,C 180,E1 -2086.721,E2 -2086.721} C_VEL
LIN {X 0,Y 573.707,Z 244.619,A -85,B 0,C 180,E1 -2086.822,E2 -2086.822} C_VEL
LIN {X 0,Y 573.82,Z 229.114,A -85,B 0,C 180,E1 -2088.753,E2 -2088.753} C_VEL
LIN {X 0,Y 574.133,Z 205.984,A -85,B 0,C 180,E1 -2091.733,E2 -2091.733} C_VEL
LIN {X 0,Y 574.413,Z 187.281,A -85,B 0,C 180,E1 -2094.196,E2 -2094.196} C_VEL
LIN {X 0,Y 573.279,Z 180.961,A -85,B 0,C 180,E1 -2095.11,E2 -2095.11} C_VEL
LIN {X 0,Y 573.255,Z 180.706,A -85,B 0,C 180,E1 -2096.19,E2 -2096.19} C_VEL
LIN {X 0,Y 573.26,Z 180.701,A -85,B 0,C 180,E1 -2099.365,E2 -2099.365} C_VEL
LIN {X 0,Y 573.25,Z 180.701,A -85,B 0,C 180,E1 -2102.228,E2 -2102.228} C_VEL
LIN {X 0,Y 573.236,Z 180.7,A -85,B 0,C 180,E1 -2104.771,E2 -2104.771} C_VEL
LIN {X 0,Y 573.25,Z 180.7,A -85,B 0,C 180,E1 -2107.165,E2 -2107.165} C_VEL
LIN {X 0,Y 573.237,Z 180.708,A -85,B 0,C 180,E1 -2109.607,E2 -2109.607} C_VEL
LIN {X 0,Y 573.237,Z 180.699,A -85,B 0,C 180,E1 -2112.641,E2 -2112.641} C_VEL
LIN {X 0,Y 573.231,Z 180.707,A -85,B 0,C 180,E1 -2115.666,E2 -2115.666} C_VEL
LIN {X 0,Y 573.24,Z 180.7,A -85,B 0,C 180,E1 -2118.544,E2 -2118.544} C_VEL
LIN {X 0,Y 573.238,Z 180.706,A -85,B 0,C 180,E1 -2121.298,E2 -2121.298} C_VEL
LIN {X 0,Y 573.26,Z 180.697,A -85,B 0,C 180,E1 -2124.011,E2 -2124.011} C_VEL
LIN {X 0,Y 573.28,Z 180.694,A -85,B 0,C 180,E1 -2126.518,E2 -2126.518} C_VEL
LIN {X 0,Y 573.234,Z 180.709,A -85,B 0,C 180,E1 -2129.115,E2 -2129.115} C_VEL
LIN {X 0,Y 573.259,Z 180.695,A -85,B 0,C 180,E1 -2131.968,E2 -2131.968} C_VEL
LIN {X 0,Y 573.248,Z 180.701,A -85,B 0,C 180,E1 -2134.589,E2 -2134.589} C_VEL
LIN {X 0,Y 573.231,Z 180.701,A -85,B 0,C 180,E1 -2137.662,E2 -2137.662} C_VEL
LIN {X 0,Y 573.271,Z 180.702,A -85,B 0,C 180,E1 -2140.728,E2 -2140.728} C_VEL
LIN {X 0,Y 573.252,Z 180.697,A -85,B 0,C 180,E1 -2143.622,E2 -2143.622} C_VEL
LIN {X 0,Y 573.234,Z 180.707,A -85,B 0,C 180,E1 -2146.529,E2 -2146.529} C_VEL
LIN {X 0,Y 573.255,Z 180.707,A -85,B 0,C 180,E1 -2148.745,E2 -2148.745} C_VEL
LIN {X 0,Y 573.284,Z 180.693,A -85,B 0,C 180,E1 -2151.54,E2 -2151.54} C_VEL
LIN {X 0,Y 573.286,Z 180.7,A -85,B 0,C 180,E1 -2154.372,E2 -2154.372} C_VEL
LIN {X 0,Y 573.303,Z 180.693,A -85,B 0,C 180,E1 -2157.892,E2 -2157.892} C_VEL
LIN {X 0,Y 573.328,Z 180.692,A -85,B 0,C 180,E1 -2160.702,E2 -2160.702} C_VEL
LIN {X 0,Y 573.233,Z 180.701,A -85,B 0,C 180,E1 -2163.514,E2 -2163.514} C_VEL
LIN {X 0,Y 573.288,Z 180.693,A -85,B 0,C 180,E1 -2165.628,E2 -2165.628} C_VEL
LIN {X 0,Y 573.283,Z 180.699,A -85,B 0,C 180,E1 -2168.459,E2 -2168.459} C_VEL
LIN {X 0,Y 573.263,Z 180.697,A -85,B 0,C 180,E1 -2171.312,E2 -2171.312} C_VEL
LIN {X 0,Y 573.267,Z 180.703,A -85,B 0,C 180,E1 -2174.193,E2 -2174.193} C_VEL
LIN {X 0,Y 573.252,Z 180.698,A -85,B 0,C 180,E1 -2177.112,E2 -2177.112} C_VEL
LIN {X 0,Y 573.244,Z 180.705,A -85,B 0,C 180,E1 -2180.077,E2 -2180.077} C_VEL
LIN {X 0,Y 573.226,Z 180.702,A -85,B 0,C 180,E1 -2183.1,E2 -2183.1} C_VEL
LIN {X 0,Y 573.251,Z 180.701,A -85,B 0,C 180,E1 -2185.41,E2 -2185.41} C_VEL
LIN {X 0,Y 573.244,Z 180.703,A -85,B 0,C 180,E1 -2188.03,E2 -2188.03} C_VEL
LIN {X 0,Y 573.225,Z 180.702,A -85,B 0,C 180,E1 -2190.883,E2 -2190.883} C_VEL
LIN {X 0,Y 573.255,Z 180.703,A -85,B 0,C 180,E1 -2193.524,E2 -2193.524} C_VEL
LIN {X 0,Y 573.234,Z 180.702,A -85,B 0,C 180,E1 -2196.05,E2 -2196.05} C_VEL
LIN {X 0,Y 573.241,Z 180.699,A -85,B 0,C 180,E1 -2198.702,E2 -2198.702} C_VEL
LIN {X 0,Y 573.223,Z 180.707,A -85,B 0,C 180,E1 -2201.593,E2 -2201.593} C_VEL
LIN {X 0,Y 573.216,Z 180.703,A -85,B 0,C 180,E1 -2204.335,E2 -2204.335} C_VEL
LIN {X 0,Y 573.235,Z 180.708,A -85,B 0,C 180,E1 -2207.359,E2 -2207.359} C_VEL
LIN {X 0,Y 573.233,Z 180.695,A -85,B 0,C 180,E1 -2210.393,E2 -2210.393} C_VEL
LIN {X 0,Y 573.247,Z 180.707,A -85,B 0,C 180,E1 -2213.078,E2 -2213.078} C_VEL
LIN {X 0,Y 573.25,Z 180.7,A -85,B 0,C 180,E1 -2215.671,E2 -2215.671} C_VEL
LIN {X 0,Y 573.231,Z 180.699,A -85,B 0,C 180,E1 -2218.185,E2 -2218.185} C_VEL
LIN {X 0,Y 573.238,Z 180.685,A -85,B 0,C 180,E1 -2220.633,E2 -2220.633} C_VEL
LIN {X 0,Y 573.208,Z 180.707,A -85,B 0,C 180,E1 -2223.023,E2 -2223.023} C_VEL
LIN {X 0,Y 573.264,Z 180.906,A -85,B 0,C 180,E1 -2223.566,E2 -2223.566} C_VEL
LIN {X 0,Y 574.741,Z 186.652,A -85,B 0,C 180,E1 -2224.273,E2 -2224.273} C_VEL
LIN {X 0,Y 574.815,Z 197.527,A -85,B 0,C 180,E1 -2225.437,E2 -2225.437} C_VEL
LIN {X 0,Y 574.379,Z 226.416,A -85,B 0,C 180,E1 -2228.465,E2 -2228.465} C_VEL
LIN {X 0,Y 574.167,Z 244.948,A -85,B 0,C 180,E1 -2230.363,E2 -2230.363} C_VEL
LIN {X 0,Y 575.198,Z 251.393,A -85,B 0,C 180,E1 -2230.504,E2 -2230.504} C_VEL
LIN {X 0,Y 574.762,Z 412.028,A -85,B 0,C 180,E1 -2232.58,E2 -2232.58} C_VEL
LIN {X 0,Y 574.642,Z 427.723,A -85,B 0,C 180,E1 -2232.931,E2 -2232.931} C_VEL
LIN {X 0,Y 574.44,Z 443.052,A -85,B 0,C 180,E1 -2233.429,E2 -2233.429} C_VEL
LIN {X 0,Y 574.264,Z 456.783,A -85,B 0,C 180,E1 -2234.017,E2 -2234.017} C_VEL
LIN {X 0,Y 574.069,Z 470.254,A -85,B 0,C 180,E1 -2234.74,E2 -2234.74} C_VEL
LIN {X 0,Y 573.859,Z 483.825,A -85,B 0,C 180,E1 -2235.632,E2 -2235.632} C_VEL
LIN {X 0,Y 573.635,Z 496.356,A -85,B 0,C 180,E1 -2236.63,E2 -2236.63} C_VEL
LIN {X 0,Y 573.477,Z 506.753,A -85,B 0,C 180,E1 -2237.616,E2 -2237.616} C_VEL
LIN {X 0,Y 573.285,Z 516.772,A -85,B 0,C 180,E1 -2238.734,E2 -2238.734} C_VEL
LIN {X 0,Y 573.243,Z 525.86,A -85,B 0,C 180,E1 -2239.939,E2 -2239.939} C_VEL
LIN {X 0,Y 573.133,Z 533.736,A -85,B 0,C 180,E1 -2241.183,E2 -2241.183} C_VEL
LIN {X 0,Y 573.074,Z 541.091,A -85,B 0,C 180,E1 -2242.602,E2 -2242.602} C_VEL
LIN {X 0,Y 573.042,Z 546.924,A -85,B 0,C 180,E1 -2244.017,E2 -2244.017} C_VEL
LIN {X 0,Y 572.951,Z 550.386,A -85,B 0,C 180,E1 -2245.075,E2 -2245.075} C_VEL
LIN {X 0,Y 573.004,Z 553.89,A -85,B 0,C 180,E1 -2246.484,E2 -2246.484} C_VEL
LIN {X 0,Y 572.938,Z 556.192,A -85,B 0,C 180,E1 -2247.891,E2 -2247.891} C_VEL
LIN {X 0,Y 572.938,Z 557.349,A -85,B 0,C 180,E1 -2249.297,E2 -2249.297} C_VEL
LIN {X 0,Y 572.938,Z 557.349,A -85,B 0,C 180,E1 -2250.703,E2 -2250.703} C_VEL
LIN {X 0,Y 572.938,Z 556.19,A -85,B 0,C 180,E1 -2252.109,E2 -2252.109} C_VEL
LIN {X 0,Y 573.004,Z 553.887,A -85,B 0,C 180,E1 -2253.516,E2 -2253.516} C_VEL
LIN {X 0,Y 572.951,Z 550.385,A -85,B 0,C 180,E1 -2254.926,E2 -2254.926} C_VEL
LIN {X 0,Y 573.014,Z 545.608,A -85,B 0,C 180,E1 -2256.338,E2 -2256.338} C_VEL
LIN {X 0,Y 573.093,Z 539.422,A -85,B 0,C 180,E1 -2257.753,E2 -2257.753} C_VEL
LIN {X 0,Y 573.135,Z 531.647,A -85,B 0,C 180,E1 -2259.173,E2 -2259.173} C_VEL
LIN {X 0,Y 573.27,Z 523.368,A -85,B 0,C 180,E1 -2260.418,E2 -2260.418} C_VEL
LIN {X 0,Y 573.386,Z 513.39,A -85,B 0,C 180,E1 -2261.668,E2 -2261.668} C_VEL
LIN {X 0,Y 573.568,Z 503.187,A -85,B 0,C 180,E1 -2262.742,E2 -2262.742} C_VEL
LIN {X 0,Y 573.743,Z 491.018,A -85,B 0,C 180,E1 -2263.82,E2 -2263.82} C_VEL
